(* CODESYS project sensata_common.library
   Company: Sensata Technologies
   DocFormat: reStructuredText
   Description: Library containing Sensata's high-level abstract modules that Sensata's other modules are built upon.
   Version: 1.0.0
   Placeholder: Sensata_Common
   Title: Sensata_Common

Project tree, tasks and I/O mapping:
  libraries: Tc2_Standard, 3.3.3.0 (Beckhoff Automation GmbH); Tc2_System, 3.4.25.0 (Beckhoff Automation GmbH); Tc2_Utilities, 3.3.52.0 (Beckhoff Automation GmbH); Tc3_JsonXml, * (Beckhoff Automation GmbH); Tc3_Module, 3.3.21.0 (Beckhoff Automation GmbH)
  Abstract/
    function block FB_Device [ST]: M_Abort, P_bAbortBusy, M_Connect, M_Disconnect, M_GetConnectStatus, P_bConnectBusy, P_bConnected, P_strDescription, P_strMake, P_strModel, P_strVersion, M_Disable, M_Enable, M_GetEnableStatus, P_bEnableBusy, P_bEnabled, M_GetPowerStatus, M_PowerOff, M_PowerOn, P_bPowerBusy, P_bPoweredOn, M_GetCurrentProgram, M_GetProgramState, M_LoadProgram, M_PauseProgram, M_StartProgram, M_StopProgram, P_bProgramControlBusy, P_enumProgramState, P_strCurrentProgram, M_Reset, P_bResetBusy
    function block FB_Machine [ST]: M_ResetCommands, M001_Aborting, M021_Clearing, M101_Stopping, M201_Resetting, M301_Starting, M321_Completing, M401_Holding, M421_Unholding, M501_Suspending, M521_Unsuspending, M_AbortStations, M_ClearStations, M_CompleteStations, M_HoldStations, M_ResetStations, M_StartStations, M_StopStations, M_SuspendStations, M_UnholdStations, M_UnsuspendStations, M_CheckStations, M_SetStation, P_arrStations
    function block FB_Module [ST]: M_ClearError, M_SetError, P_bError, P_strErrorMessage, P_udintErrorCode, M_Log, M_LogError, M_LogMessage, M_LogWarning, P_bLoggingEnabled, P_strUniqueId
    function block FB_StateMachine [ST]: P_bAbortable, P_bStoppable, P_enumState, M_Abort, M_Clear, M_Complete, M_Hold, M_Reset, M_Start, M_Stop, M_Suspend, M_Unhold, M_Unsuspend, A000_Aborting_Entry, A001_Aborting, A002_Aborting_Exit, M000_Aborting_Entry, M001_Aborting, M002_Aborting_Exit, A010_Aborted_Entry, A011_Aborted, A012_Aborted_Exit, M010_Aborted_Entry, M011_Aborted, M012_Aborted_Exit, A020_Clearing_Entry, A021_Clearing, A022_Clearing_Exit, M020_Clearing_Entry, M021_Clearing, M022_Clearing_Exit, A100_Stopping_Entry, A101_Stopping, A102_Stopping_Exit, M100_Stopping_Entry, M101_Stopping, M102_Stopping_Exit, A110_Stopped_Entry, A111_Stopped, A112_Stopped_Exit, M110_Stopped_Entry, M111_Stopped, M112_Stopped_Exit, A200_Resetting_Entry, A201_Resetting, A202_Resetting_Exit, M200_Resetting_Entry, M201_Resetting, M202_Resetting_Exit, A210_Idle_Entry, A211_Idle, A212_Idle_Exit, M210_Idle_Entry, M211_Idle, M212_Idle_Exit, A300_Starting_Entry, A301_Starting, A302_Starting_Exit, M300_Starting_Entry, M301_Starting, M302_Starting_Exit, A310_Execute_Entry, A311_Execute, A312_Execute_Exit, M310_Execute_Entry, M311_Execute, M312_Execute_Exit, A320_Completing_Entry, A321_Completing, A322_Completing_Exit, M320_Completing_Entry, M321_Completing, M322_Completing_Exit, A330_Complete_Entry, A331_Complete, A332_Complete_Exit, M330_Complete_Entry, M331_Complete, M332_Complete_Exit, A400_Holding_Entry, A401_Holding, A402_Holding_Exit, M400_Holding_Entry, M401_Holding, M402_Holding_Exit, A410_Held_Entry, A411_Held, A412_Held_Exit, M410_Held_Entry, M411_Held, M412_Held_Exit, A420_Unholding_Entry, A421_Unholding, A422_Unholding_Exit, M420_Unholding_Entry, M421_Unholding, M422_Unholding_Exit, A500_Suspending_Entry, A501_Suspending, A502_Suspending_Exit, M500_Suspending_Entry, M501_Suspending, M502_Suspending_Exit, A510_Suspended_Entry, A511_Suspended, A512_Suspended_Exit, M510_Suspended_Entry, M511_Suspended, M512_Suspended_Exit, A520_Unsuspending_Entry, A521_Unsuspending, A522_Unsuspending_Exit, M520_Unsuspending_Entry, M521_Unsuspending, M522_Unsuspending_Exit, A_StateMachine
    function block FB_Station [ST]: M001_Aborting, M021_Clearing, M101_Stopping, M201_Resetting, M301_Starting, M321_Completing, M401_Holding, M421_Unholding, M501_Suspending, M521_Unsuspending, M_AbortDevices, M_CheckForDeviceErrors, M_ClearDevices, M_CompleteDevices, M_HoldDevices, M_ResetDevices, M_StartDevices, M_StopDevices, M_SuspendDevices, M_UnholdDevices, M_UnsuspendDevices, M_SetDevice, P_arrDevices, M_Init, FB_exit
  Concrete/
    Obsolete/
      function block FB_DeviceTestStation_Old [ST]: M000_Aborting_Entry, M001_Aborting, M002_Aborting_Exit, M010_Aborted_Entry, M011_Aborted, M012_Aborted_Exit, M020_Clearing_Entry, M021_Clearing, M022_Clearing_Exit, M100_Stopping_Entry, M101_Stopping, M102_Stopping_Exit, M110_Stopped_Entry, M111_Stopped, M112_Stopped_Exit, M200_Resetting_Entry, M201_Resetting, M202_Resetting_Exit, M210_Idle_Entry, M211_Idle, M212_Idle_Exit, M300_Starting_Entry, M301_Starting, M302_Starting_Exit, M310_Execute_Entry, M311_Execute, M312_Execute_Exit, M320_Completing_Entry, M321_Completing, M322_Completing_Exit, M330_Complete_Entry, M331_Complete, M332_Complete_Exit, M400_Holding_Entry, M401_Holding, M402_Holding_Exit, M410_Held_Entry, M411_Held, M412_Held_Exit, M420_Unholding_Entry, M421_Unholding, M422_Unholding_Exit, M500_Suspending_Entry, M501_Suspending, M502_Suspending_Exit, M510_Suspended_Entry, M511_Suspended, M512_Suspended_Exit, M520_Unsuspending_Entry, M521_Unsuspending, M522_Unsuspending_Exit, A_DeviceTestTracking
    function block FB_DeviceController [ST]: M_Init, M00_Abort, M02_Clear, M10_Stop, M20_Reset, M30_Start, M32_Complete, M40_Hold, M42_Unhold, M50_Suspend, M52_Unsuspend
    function block FB_DeviceTestStation [ST]: A_DeviceTestTracking
    function block FB_SimpleMachine [ST]: A_Buttons, A_RunSimpleMachine, A_StopAndAbort, M011_Aborted, M111_Stopped, M211_Idle, M311_Execute, M331_Complete, M411_Held, M511_Suspended
    function block FB_SimpleStation [ST]: A_Buttons, A_RunSimpleStation, A_StopAndAbort, M011_Aborted, M111_Stopped, M211_Idle, M311_Execute, M331_Complete, M411_Held, M511_Suspended
    function block FB_StandardStation [ST]: M_AwaitCycleEnd, M_AwaitCycleStart, M_ClearUserPrompt, M_HandleException, M_ResetCycle, M_SetUserPrompt
  Enumerators/
    data type E_DeviceControllerError
    data type E_MachineError
    data type E_PackMLState
    data type E_ProgramState
    data type E_StationError
  Global Variable Lists/
    global variables GVL_Constants
  Interfaces/
    Devices/
      interface I_Abortable: M_Abort, P_bAbortBusy
      interface I_Connectable: M_Connect, M_Disconnect, M_GetConnectStatus, P_bConnectBusy, P_bConnected
      interface I_DeviceInfo: P_strDescription, P_strMake, P_strModel, P_strVersion
      interface I_Enableable: M_Disable, M_Enable, M_GetEnableStatus, P_bEnableBusy, P_bEnabled
      interface I_Powerable: M_GetPowerStatus, M_PowerOff, M_PowerOn, P_bPowerBusy, P_bPoweredOn
      interface I_Programmable: M_GetCurrentProgram, M_GetProgramState, M_LoadProgram, M_PauseProgram, M_StartProgram, M_StopProgram, P_bProgramControlBusy, P_enumProgramState, P_strCurrentProgram
      interface I_Resettable: M_Reset, P_bResetBusy
    Machines/
      interface I_MachineStationStateControl: M_AbortStations, M_ClearStations, M_CompleteStations, M_HoldStations, M_ResetStations, M_StartStations, M_StopStations, M_SuspendStations, M_UnholdStations, M_UnsuspendStations
    Modules/
      interface I_ErrorHandling: M_ClearError, M_SetError, P_bError, P_strErrorMessage, P_udintErrorCode
      interface I_Logging: M_LogError, M_LogMessage, M_LogWarning, P_bLoggingEnabled
    State Machine/
      Stateful/
        interface I_ExecuteStateOnly: M310_Execute_Entry, M312_Execute_Exit
        interface I_SimpleExecuteStateOnly: M311_Execute
        interface I_SimpleStateful
        interface I_SimpleTransitionStatesOnly: M001_Aborting, M021_Clearing, M101_Stopping, M201_Resetting, M301_Starting, M321_Completing, M401_Holding, M421_Unholding, M501_Suspending, M521_Unsuspending
        interface I_SimpleWaitingStatesOnly: M011_Aborted, M111_Stopped, M211_Idle, M331_Complete, M411_Held, M511_Suspended
        interface I_Stateful
        interface I_TransitionStatesOnly: M000_Aborting_Entry, M002_Aborting_Exit, M020_Clearing_Entry, M022_Clearing_Exit, M100_Stopping_Entry, M102_Stopping_Exit, M200_Resetting_Entry, M202_Resetting_Exit, M300_Starting_Entry, M302_Starting_Exit, M320_Completing_Entry, M322_Completing_Exit, M400_Holding_Entry, M402_Holding_Exit, M420_Unholding_Entry, M422_Unholding_Exit, M500_Suspending_Entry, M502_Suspending_Exit, M520_Unsuspending_Entry, M522_Unsuspending_Exit
        interface I_WaitingStatesOnly: M010_Aborted_Entry, M012_Aborted_Exit, M110_Stopped_Entry, M112_Stopped_Exit, M210_Idle_Entry, M212_Idle_Exit, M310_Execute_Entry, M312_Execute_Exit, M330_Complete_Entry, M332_Complete_Exit, M410_Held_Entry, M412_Held_Exit, M510_Suspended_Entry, M512_Suspended_Exit
      interface I_StateControl: M_Abort, M_Clear, M_Complete, M_Hold, M_Reset, M_Start, M_Stop, M_Suspend, M_Unhold, M_Unsuspend
    Stations/
      interface I_StationDeviceControl: M_AbortDevices, M_ClearDevices, M_CompleteDevices, M_HoldDevices, M_ResetDevices, M_StartDevices, M_StopDevices, M_SuspendDevices, M_UnholdDevices, M_UnsuspendDevices
  Project Information/
    function F_GetCompany [ST]
    function F_GetTitle [ST]
    function F_GetVersion [ST]
  Structs/
    data type ST_Prompt
  Types/
    data type T_MachineStationArray
    data type T_StationDeviceArray
  Version/
    global variables Global_Version
*)

// Enumerators/E_DeviceControllerError
{attribute 'qualified_only'}
{attribute 'strict'}
{attribute 'qualified_only'}
TYPE E_DeviceControllerError :
(
	None := 0,
	ClearError := 0200,
	StopError := 1000,
	ResetError := 2000,
	StartError := 3000,
	CompleteError := 3200,
	HoldError := 4000,
	UnholdError := 4200,
	SuspendError := 5000,
	UnsuspendError := 5200
) UDINT;
END_TYPE

// Enumerators/E_MachineError
{attribute 'qualified_only'}
{attribute 'strict'}
TYPE E_MachineError :
(
	None := 0,
	
	StationError := 100
) UDINT;
END_TYPE

// Enumerators/E_PackMLState
(* Represents all possible PackML states. *)
{attribute 'qualified_only'}
{attribute 'strict'}
{attribute 'to_string'}
TYPE E_PackMLState :
(
	None := -1,
	Aborting := 00, 
	Aborted := 01,
	Clearing := 02,
	Stopping := 10,
	Stopped := 11,
	Resetting := 20,
	Idle := 21, 
	Starting := 30,
	Execute := 31,
	Completing := 32,
	Complete := 33,
	Holding := 40,
	Held := 41,
	Unholding := 42,
	Suspending := 50,
	Suspended := 51,
	Unsuspending := 52
) := None;
END_TYPE

// Enumerators/E_ProgramState
(*
The possible states for a program loaded on a device.
*)
{attribute 'qualified_only'}
{attribute 'strict'}
{attribute 'to_string'}
TYPE E_ProgramState :
(
	(* The unknown state means that the current program state is not known.
		This is the default enumerator state. *)
	Unknown := 0,
	
	(* A program that is stopped means that, when started, the program would begin
		from the start. Going from the Running state to the Stopped state or from
		the Paused state to the Stopped state will reset the program execution
		back to the beginning. *)
	Stopped,
	
	(* A program in the running state is actively executing. Going from the
		Stopped state to the Running state will begin execution from the
		beginning of the program, and going from the Paused state to the
		Running state will continue execution from whichever point it was
		at when the transition from Running to Paused occurred.*)
	Running,
	
	(* A program that is paused is not executing, but is also not reset to the
		start. When going from the Running state to the Paused state, the
		program execution is held in the state it was in when the transition
		occurred. *)
	Paused
);
END_TYPE

// Enumerators/E_StationError
{attribute 'qualified_only'}
{attribute 'strict'}
(*
Errors for use in FB_Station
*)
TYPE E_StationError :
(
	None			:= 000000000,
	
	DeviceError		:= 301000000
) UDINT;
END_TYPE

// Structs/ST_Prompt
TYPE ST_Prompt :
STRUCT
	(* Code for this prompt message. *)
	udintCode: UDINT;
	(* Default message text (for debug and if localization not used) *)
	strMessage: T_MaxString;
END_STRUCT
END_TYPE

// Types/T_MachineStationArray
(* Alias for an array of pointers to stations. *)
TYPE T_MachineStationArray : 
	ARRAY[1..GVL_Constants.uintMAX_MACHINE_STATION_COUNT] 
		OF POINTER TO FB_Station;
END_TYPE

// Types/T_StationDeviceArray
(* Alias for an array of pointers to devices. *)
TYPE T_StationDeviceArray :
	ARRAY[1..GVL_Constants.uintMAX_STATION_DEVICE_COUNT]
		OF POINTER TO FB_DeviceController;
END_TYPE

// Global Variable Lists/GVL_Constants
{attribute 'qualified_only'}
VAR_GLOBAL CONSTANT
	uintMAX_STATION_DEVICE_COUNT : UINT := 32;
	uintMAX_MACHINE_STATION_COUNT : UINT := 32;
END_VAR

// Version/Global_Version
{attribute 'TcGenerated'}
{attribute 'no-analysis'}
{attribute 'linkalways'}
// This function has been automatically generated from the project information.
VAR_GLOBAL CONSTANT
	{attribute 'const_non_replaced'}
	stLibVersion_Sensata_Common : ST_LibVersion := (iMajor := 1, iMinor := 0, iBuild := 0, iRevision := 0, nFlags := 0, sVersion := '1.0.0');
END_VAR

// Abstract/FB_Device
(*
===============================================================================
Device
===============================================================================
:Contact: Kevin Sanita <ksanita@sensata.com>
:Last Edited: December 2021

:Description: Parent class for all devices in the Sensata libraries.

:Notes:
* Devices are defined as physical objects that the PAC must control or communicate with.
* All children of this Device class should implement ``I_DeviceInfo`` to easily import the required properties.
* Ensure the device properties are properly implemented and kept up to date if a device is updated.

:Change Log:
- **December 2021** Initial version
*)
{attribute 'hide_all_locals'}
FUNCTION_BLOCK ABSTRACT FB_Device EXTENDS FB_Module 
	IMPLEMENTS 
		I_DeviceInfo, // Device information
		I_Abortable, // Some devices may need to perform specific tasks when aborted
		I_Connectable, // Connecting and disconnecting is a common functionality of devices
		I_Enableable, // Many devices can be enabled/disabled without necessarily changing state
		I_Powerable, // Many devices need a specific command in order to energize
		I_Programmable, // Managing programs is a common functionality of devices with internal logic
		I_Resettable // Devices often need a reset command to clear any errors
VAR_INPUT		
END_VAR
VAR_OUTPUT
END_VAR
VAR
	dev_bConnected: BOOL; // TRUE if the device is connected
	dev_bEnabled: BOOL; // TRUE if the device is enabled
	dev_enumProgramState: E_ProgramState; // Current control state
	dev_bPoweredOn: BOOL; // TRUE if the device is powered on
	dev_strCurrentProgram: STRING(255); // Current program
END_VAR

(* Performs tasks that should be performed when the device is aborted. *)
METHOD M_Abort : BOOL
M_Abort := TRUE;
THIS^.M_LogWarning('M_Abort not implemented!');

IF NOT THIS^.P_bError THEN
	THIS^.M_SetError(16#FFFF, 'Aborted!');
END_IF
END_METHOD

(* True while aborting, false otherwise. *)
PROPERTY P_bAbortBusy : BOOL
GET
P_bAbortBusy := FALSE;
END_GET
END_PROPERTY

(* Connect to the device. *)
METHOD M_Connect : BOOL
dev_bConnected := TRUE;
M_Connect := TRUE;
THIS^.M_LogWarning('M_Connect not implemented!');
END_METHOD

(* Disconnect from the camera. *)
METHOD M_Disconnect : BOOL
dev_bConnected := FALSE;
M_Disconnect := TRUE;
THIS^.M_LogWarning('M_Disconnect not implemented!');
END_METHOD

(* Get the device connection status. *)
METHOD M_GetConnectStatus : BOOL
VAR_OUTPUT
	(* TRUE if the device is connected, FALSE otherwise. *)
	bConnected	: BOOL;
END_VAR
bConnected := THIS^.dev_bConnected;
M_GetConnectStatus := TRUE;
END_METHOD

(* TRUE while the device is connecting or disconnecting. *)
PROPERTY P_bConnectBusy : BOOL
GET
P_bConnectBusy := FALSE;
END_GET
END_PROPERTY

(* TRUE if the camera is connected. *)
PROPERTY P_bConnected : BOOL
GET
P_bConnected := dev_bConnected;
END_GET
END_PROPERTY

(*
A brief description of the device.
*)
PROPERTY P_strDescription : T_MaxString
GET
END_GET
END_PROPERTY

(*
The manufacturer of the device.
*)
PROPERTY P_strMake : T_MaxString
GET
END_GET
END_PROPERTY

(*
The model name or ID of the device.
*)
PROPERTY P_strModel : T_MaxString
GET
END_GET
END_PROPERTY

(*
The version(s) of the device that the function block supports.
*)
PROPERTY P_strVersion : T_MaxString
GET
END_GET
END_PROPERTY

(* Disable the device. *)
METHOD M_Disable : BOOL
dev_bEnabled := FALSE;
M_Disable := TRUE;
THIS^.M_LogWarning('M_Disable is not implemented!');
END_METHOD

(* Enable the device *)
METHOD M_Enable : BOOL
dev_bEnabled := TRUE;
M_Enable := TRUE;
THIS^.M_LogWarning('M_Enable is not implemented!');
END_METHOD

(* Get the current enable status of the device. *)
METHOD M_GetEnableStatus : BOOL
VAR_OUTPUT
	bEnabled	: BOOL;
END_VAR
bEnabled := THIS^.dev_bEnabled;
M_GetEnableStatus := TRUE;
END_METHOD

(* TRUE while the device is busy enabling or disabling. *)
PROPERTY P_bEnableBusy : BOOL
GET
END_GET
END_PROPERTY

(* TRUE if the device is enabled. *)
PROPERTY P_bEnabled : BOOL
GET
P_bEnabled := dev_bEnabled;
END_GET
END_PROPERTY

(* Gets the current power status of the device. *)
METHOD M_GetPowerStatus : BOOL
VAR_OUTPUT
	bPoweredOn	: BOOL;
END_VAR
bPoweredOn := THIS^.dev_bPoweredOn;
M_GetPowerStatus := TRUE;
END_METHOD

(*
Power off the device or module
*)
METHOD M_PowerOff : BOOL
dev_bPoweredOn := FALSE;
M_PowerOff := TRUE;
THIS^.M_LogWarning('M_PowerOff is not implemented!');
END_METHOD

(*
Power on the device or module.
*)
METHOD M_PowerOn : BOOL
dev_bPoweredOn := TRUE;
M_PowerOn := TRUE;
THIS^.M_LogWarning('M_PowerOn is not implemented!');
END_METHOD

(* TRUE while the device is powering on or off. *)
PROPERTY P_bPowerBusy : BOOL
GET
P_bPowerBusy := FALSE;
END_GET
END_PROPERTY

(*
TRUE if the module or device is powered on.
*)
PROPERTY P_bPoweredOn : BOOL
GET
P_bPoweredOn := dev_bPoweredOn;
END_GET
END_PROPERTY

(* Gets the program currently loaded on the device. *)
METHOD M_GetCurrentProgram : BOOL
VAR_OUTPUT
	strCurrentProgram	: Tc2_System.T_MaxString;
END_VAR
strCurrentProgram := THIS^.dev_strCurrentProgram;
M_GetCurrentProgram := TRUE;
END_METHOD

(* Gets the current control state. *)
METHOD M_GetProgramState : BOOL
VAR_OUTPUT
	enumProgramState	: E_ProgramState;
END_VAR
enumProgramState := THIS^.dev_enumProgramState;
M_GetProgramState := TRUE;
END_METHOD

(* Load a new program. *)
METHOD M_LoadProgram : BOOL
VAR_INPUT
END_VAR
dev_strCurrentProgram := '';
M_LoadProgram := TRUE;
THIS^.M_LogWarning('M_LoadProgram not implemented!');
END_METHOD

(* Pauses the camera program. *)
METHOD M_PauseProgram : BOOL
dev_enumProgramState := E_ProgramState.Paused;
M_PauseProgram := TRUE;
THIS^.M_LogWarning('M_PauseProgram not implemented!');
END_METHOD

(* Starts the camera program. *)
METHOD M_StartProgram : BOOL
dev_enumProgramState := E_ProgramState.Running;
M_StartProgram := TRUE;
THIS^.M_LogWarning('M_StartProgram not implemented!');
END_METHOD

(* Stops the camera program. *)
METHOD M_StopProgram : BOOL
dev_enumProgramState := E_ProgramState.Stopped;
M_StopProgram := TRUE;
THIS^.M_LogWarning('M_StopProgram not implemented!');
END_METHOD

(*
TRUE while a program is being loaded
*)
PROPERTY P_bProgramControlBusy : BOOL
GET
P_bProgramControlBusy := FALSE;
END_GET
END_PROPERTY

(* Current device program state. *)
PROPERTY P_enumProgramState : E_ProgramState
GET
P_enumProgramState := dev_enumProgramState;
END_GET
END_PROPERTY

(* Current program. *)
PROPERTY P_strCurrentProgram : Tc2_System.T_MaxString
GET
P_strCurrentProgram := dev_strCurrentProgram;
END_GET
END_PROPERTY

(* Resets the device and clears any external errors. *)
METHOD M_Reset : BOOL
M_Reset := TRUE;
THIS^.M_ClearError();
THIS^.M_LogWarning('M_Reset not implemented!');
END_METHOD

(* Stays high while module is resetting. *)
PROPERTY P_bResetBusy : BOOL
GET
P_bResetBusy := FALSE;
END_GET
END_PROPERTY

END_FUNCTION_BLOCK

// Interfaces/Devices/I_DeviceInfo
(*
===============================================================================
Device Information
===============================================================================

:Description: Contains the standard properties of the Device function block for easier implementation.

*)
INTERFACE I_DeviceInfo

PROPERTY P_strDescription : T_MaxString
GET
END_GET
END_PROPERTY

PROPERTY P_strMake : T_MaxString
GET
END_GET
END_PROPERTY

PROPERTY P_strModel : T_MaxString
GET
END_GET
END_PROPERTY

PROPERTY P_strVersion : T_MaxString
GET
END_GET
END_PROPERTY

END_INTERFACE

// Abstract/FB_Module
(*
===============================================================================
Module
===============================================================================
:Contact: Kevin Sanita <ksanita@sensata.com>
:Last Edited: December 2021

:Description: All function blocks in Sensata libraries must derive from this. Handles basic functions like errors and logging. 

:Notes:
* You can use ``M_LogError``, ``M_LogWarning``, and ``M_LogMessage`` to output string messages to the "Error list" in Visual Studio
* ``M_SetError`` and ``M_ClearError`` can be used to set an error with a specified error code and message and then clear said error.
* You can use ``P_bError``, ``P_strErrorMessage`` and ``P_udintErrorCode`` to access error information.

:Change Log:
- **December 2021** Initial version

*)
FUNCTION_BLOCK ABSTRACT FB_Module
	IMPLEMENTS
		I_ErrorHandling, // All modules have error handling
		I_Logging // All modules have logging
VAR_INPUT CONSTANT
	in_strUniqueId : T_MaxString; (* A unique name for this function block to be used in logging. *)
	in_bDisableLogging: BOOL; (* Set TRUE to disable all logging. *)
END_VAR
VAR_OUTPUT
END_VAR
VAR
	mod_bError : BOOL; (* TRUE if there is an error. *)
	mod_udintErrorCode : UDINT; (* 0 if no error, error code otherwise. Refer to module-specific documentation for code meaning. *)
	mod_strErrorMessage : T_MaxString; (* Blank if no error, error message otherwise. *)
	mod_bLoggingEnabled: BOOL := TRUE; (* Enables and disabled logging. *)
END_VAR

(*
Clears the current error. Sets P_bError to false, P_strErrorMessage to blank, and P_udintErrorCode to zero.
*)
METHOD M_ClearError : BOOL
IF THIS^.mod_bError THEN
	THIS^.M_LogMessage('Error cleared.');
END_IF

THIS^.mod_bError := FALSE;
THIS^.mod_udintErrorCode := 0;
THIS^.mod_strErrorMessage := '';

M_ClearError := TRUE;
END_METHOD

(*
Sets an error with the given code and message.
*)
METHOD M_SetError : BOOL
VAR_INPUT
	udintErrorCode : UDINT; (* Error codes are specific to the concrete modules. Check documentation of the module for error code meaning. *)
	strErrorMessage : T_MaxString; (* Error messages should be short, but descriptive enough to still be useful. *)
END_VAR
// If there is not already an error set or error code or message is different,
// update the values and print to log
IF (NOT mod_bError) 
		OR (mod_udintErrorCode <> udintErrorCode)
		OR (mod_strErrorMessage <> strErrorMessage) THEN
	THIS^.mod_bError := TRUE;
	THIS^.mod_udintErrorCode := udintErrorCode;
	THIS^.mod_strErrorMessage := strErrorMessage;
	THIS^.M_LogError(strErrorMessage);
END_IF
END_METHOD

(*
TRUE if there is an error, FALSE otherwise.
*)
PROPERTY P_bError : BOOL
GET
P_bError := mod_bError;
END_GET
END_PROPERTY

(*
A description of the current error. Will be blank if no error.
*)
PROPERTY P_strErrorMessage : Tc2_System.T_MaxString
GET
P_strErrorMessage := mod_strErrorMessage;
END_GET
END_PROPERTY

(*
The ID of the current error. Review module-specific documentation for meaning of error codes. Will be 0 if no error.
*)
PROPERTY P_udintErrorCode : UDINT
GET
P_udintErrorCode := mod_udintErrorCode;
END_GET
END_PROPERTY

METHOD PRIVATE M_Log : BOOL
VAR_INPUT
	strMessage : T_MaxString;
	dwordMsgCtrlMask : DWORD;
END_VAR
VAR
	fbFormat: FB_FormatString;
END_VAR
// If logging is enabled, print to ADS log
IF NOT in_bDisableLogging THEN
	// Format the message with the unique ID
	fbFormat(
		sFormat:= '%s --- %s', 
		arg1:= F_STRING(in_strUniqueId), 
		arg2:= F_STRING(strMessage));
	
	// Return false if there was a format error
	IF fbFormat.bError THEN
		M_Log := FALSE;
	ELSE
		// Log the message to ADS
		ADSLOGSTR(
			msgCtrlMask:= dwordMsgCtrlMask,
			msgFmtStr:= '%s',
			strArg:= fbFormat.sOut);
		M_Log := TRUE;
	END_IF
// If logging is not enabled, don't do anything
ELSE
	M_Log := TRUE;
END_IF
END_METHOD

(*
Prints an error message to the Error List in Visual Studio.
*)
METHOD M_LogError : BOOL
VAR_INPUT
	strMessage : T_MaxString;
END_VAR
M_LogError := M_Log(strMessage, ADSLOG_MSGTYPE_ERROR OR ADSLOG_MSGTYPE_LOG);
END_METHOD

(*
Outputs a message to the Error List in Visual Studio
*)
METHOD M_LogMessage : BOOL
VAR_INPUT
	strMessage : T_MaxString;
END_VAR
M_LogMessage := M_Log(strMessage, ADSLOG_MSGTYPE_HINT OR ADSLOG_MSGTYPE_LOG);
END_METHOD

(*
Outputs a warning message to the Error List in Visual Studio
*)
METHOD M_LogWarning : BOOL
VAR_INPUT
	strMessage : T_MaxString;
END_VAR
M_LogWarning := M_Log(strMessage, ADSLOG_MSGTYPE_WARN OR ADSLOG_MSGTYPE_LOG);
END_METHOD

(* TRUE when ADS logging is enabled, false otherwise. *)
PROPERTY P_bLoggingEnabled : BOOL
GET
P_bLoggingEnabled := NOT in_bDisableLogging;
END_GET
END_PROPERTY

PROPERTY P_strUniqueId : T_MaxString
GET
P_strUniqueId := in_strUniqueId;
END_GET
END_PROPERTY

END_FUNCTION_BLOCK

// Interfaces/Modules/I_ErrorHandling
INTERFACE I_ErrorHandling

(*
Clears the current error. Sets P_bError to false, P_strErrorMessage to blank, and P_udintErrorCode to zero.
*)
METHOD M_ClearError : BOOL
END_METHOD

(*
Sets an error with the given code and message.
*)
METHOD M_SetError : BOOL
VAR_INPUT
	udintErrorCode : UDINT; (* Error codes are specific to the concrete modules. Check documentation of the module for error code meaning. *)
	strErrorMessage : T_MaxString; (* Error messages should be short, but descriptive enough to still be useful. *)
END_VAR
END_METHOD

(*
TRUE if there is an error, FALSE otherwise.
*)
PROPERTY P_bError : BOOL
GET
END_GET
END_PROPERTY

(*
A description of the current error. Will be blank if no error.
*)
PROPERTY P_strErrorMessage : Tc2_System.T_MaxString
GET
END_GET
END_PROPERTY

(*
The ID of the current error. Review module-specific documentation for meaning of error codes. Will be 0 if no error.
*)
PROPERTY P_udintErrorCode : UDINT
GET
END_GET
END_PROPERTY

END_INTERFACE

// Interfaces/Modules/I_Logging
INTERFACE I_Logging

(*
Prints an error message to the Error List in Visual Studio.
*)
METHOD M_LogError : BOOL
VAR_INPUT
	strMessage : T_MaxString;
END_VAR
END_METHOD

(*
Outputs a message to the Error List in Visual Studio
*)
METHOD M_LogMessage : BOOL
VAR_INPUT
	strMessage : T_MaxString;
END_VAR
END_METHOD

(*
Outputs a warning message to the Error List in Visual Studio
*)
METHOD M_LogWarning : BOOL
VAR_INPUT
	strMessage : T_MaxString;
END_VAR
END_METHOD

(* TRUE when ADS logging is enabled, false otherwise. *)
PROPERTY P_bLoggingEnabled : BOOL
GET
END_GET
END_PROPERTY

END_INTERFACE

// Interfaces/Devices/I_Abortable
(*
===============================================================================
Abortable
===============================================================================

:Description: Implements the ability to quickly and safely abort the device.
*)
INTERFACE I_Abortable

(* This method should rapidly but safely abort the device and set an error
	indicating that the device has been aborted. Method should return TRUE
	once successfully aborted and false otherwise. *)
METHOD M_Abort : BOOL
VAR_INPUT
END_VAR
END_METHOD

(* This property should be TRUE while any method in this interface is actively
	executing, or FALSE otherwise. *)
PROPERTY P_bAbortBusy : BOOL
GET
END_GET
END_PROPERTY

END_INTERFACE

// Interfaces/Devices/I_Connectable
(*
===============================================================================
Connectable
===============================================================================

:Description: Implements the ability to send explicit connect and disconnect
	commands to the device.
*)
INTERFACE I_Connectable

(* This method should establish any external connections required to use the
	functions of the device, and return TRUE and set P_bConnected to TRUE once
	connected. *)
METHOD M_Connect : BOOL
VAR_INPUT
END_VAR
END_METHOD

(* This method should break any connections established by M_Connect. It should
	immediately set P_bConnected to false unless all connections are known to
	be still active, and return TRUE once those connections are all fully
	disconnected. *)
METHOD M_Disconnect : BOOL
VAR_INPUT
END_VAR
END_METHOD

(* This method should explicitly check the connection status of the device.
	Once the connection status is known, this method should return TRUE.
	If this method fails, P_bConnected should be set to FALSE since the device
	is not absolutely known to still be connected. *)
METHOD M_GetConnectStatus : BOOL
VAR_INPUT
END_VAR
VAR_OUTPUT
	(* This should return TRUE if all connections required to make the device
		function properly are known to be connected, and FALSE otherwise. *)
	bConnected : BOOL;
END_VAR
END_METHOD

(* This property should be TRUE while any method in this interface is actively
	executing, or FALSE otherwise. *)
PROPERTY P_bConnectBusy : BOOL
GET
END_GET
END_PROPERTY

(* This should be set to TRUE if M_Connect is successful or M_GetConnectStatus
	determines the device to be connected, and set to FALSE if M_Disconnect is
	called at all, M_GetConnectStatus fails, or M_GetConnectStatus determines
	the device to be not connected. *)
PROPERTY P_bConnected : BOOL
GET
END_GET
END_PROPERTY

END_INTERFACE

// Interfaces/Devices/I_Enableable
(*
===============================================================================
Enableable
===============================================================================

:Description: Interface that implements the ability for the device to enable to
	(and disable from) a ready-to-start state from an energized state.

*)
INTERFACE I_Enableable

(* This method should return to the device to the state it was prior to being
	enabled. P_bEnabled should be immediately set to false unless the status of
	the device is explicitly known to still be enabled. After being disabled,
	the device should typically be unable to perform process steps. Once
	successfully disabled, this method should return TRUE. *)
METHOD M_Disable : BOOL
VAR_INPUT
END_VAR
END_METHOD

(* This method should perform any tasks that must be performed after a device
	is energized, but prior to the device being used in a process, and then
	return TRUE and set P_bEnabled to TRUE once those tasks are completed. *)
METHOD M_Enable : BOOL
VAR_INPUT
END_VAR
END_METHOD

(* This method should explicitly check the enable status of the device.
	Once the enable status is known, this method should return TRUE.
	If this method fails, P_bEnabled should be set to FALSE since the device
	is not absolutely known to still be enabled. *)
METHOD M_GetEnableStatus : BOOL
VAR_INPUT
END_VAR
VAR_OUTPUT
	(* This should return TRUE if the device is explicitly known to be
		enabled, or FALSE otherwise. *)
	bEnabled : BOOL;
END_VAR
END_METHOD

(* This property should be TRUE while any method in this interface is actively
	executing, or FALSE otherwise. *)
PROPERTY P_bEnableBusy : BOOL
GET
END_GET
END_PROPERTY

(* This should be set to TRUE if M_Enable is successful or M_GetEnableStatus
	determines the device to be enabled, and set to FALSE if M_Disable is
	called at all, M_GetEnableStatus fails, or M_GetEnableStatus determines
	the device to be not enabled. *)
PROPERTY P_bEnabled : BOOL
GET
END_GET
END_PROPERTY

END_INTERFACE

// Interfaces/Devices/I_Powerable
(*
===============================================================================
Powerable
===============================================================================

:Description: Interface that implements the ability to energize and de-energize
	a device. 

*)
INTERFACE I_Powerable

(* This method should explicitly check the power status of the device.
	Once the power status is known, this method should return TRUE.
	If this method fails, P_bPoweredOn should be set to FALSE since the device
	is not absolutely known to still be powered on. *)
METHOD M_GetPowerStatus : BOOL
VAR_INPUT
END_VAR
VAR_OUTPUT
	(* This should return TRUE if the device is explicitly known to be
		powered on, or FALSE otherwise. *)
	bPoweredOn : BOOL;
END_VAR
END_METHOD

(* This method should de-energize the device and then return TRUE once
	successful. P_bPoweredOn should be set to FALSE immediately when this is
	called unless the device is explicitly known to still be powered on. *)
METHOD M_PowerOff : BOOL
VAR_INPUT
END_VAR
END_METHOD

(* This method should energize the device and then return TRUE and set
	P_bPoweredOn to TRUE once successful. *)
METHOD M_PowerOn : BOOL
VAR_INPUT
END_VAR
END_METHOD

(* This property should be TRUE while any method in this interface is actively
	executing, or FALSE otherwise. *)
PROPERTY P_bPowerBusy : BOOL
GET
END_GET
END_PROPERTY

(* This should be set to TRUE if M_PowerOn is successful or if M_GetPowerStatus
	determines that the device is powered on. Otherwise, this should be FALSE. *)
PROPERTY P_bPoweredOn : BOOL
GET
END_GET
END_PROPERTY

END_INTERFACE

// Interfaces/Devices/I_Programmable
(*
===============================================================================
Programmable
===============================================================================

:Description: Interface that implements the ability to manage devices that have
	internally-defined execution programs that can be loaded and/or controlled
	by an external source.

:Change Log:
* June 2022 - Change P_bProgramLoading to P_bProgramBusy
*)
INTERFACE I_Programmable

(* This method should explicitly get the current program loaded on the device.
	If the current program is successfully gotten, this method should return
	TRUE and set P_strCurrentProgram and strCurrentProgram to the gotten
	program name. If this method fails, both should be set to empty strings. *)
METHOD M_GetCurrentProgram : BOOL
VAR_INPUT
END_VAR
VAR_OUTPUT
	(* This should be set to the name of the currently loaded program if
		the method was successful, or a blank string otherwise. *)
	strCurrentProgram : T_MaxString;
END_VAR
END_METHOD

(* This method should explicitly check the program state of the device.
	Once the program state is known, this method should return TRUE and set
	P_enumProgramState and enumProgramState to the relevant E_ProgramState
	value, else it should set both to E_ProgramState.Unknown. *)
METHOD M_GetProgramState : BOOL
VAR_INPUT
END_VAR
VAR_OUTPUT
	(* If the program state is successfully gotten, this should be set to
		the relevant E_ProgramState value. If this method fails, this should
		be set to E_ProgramState.Unknown. *)
	enumProgramState : E_ProgramState;
END_VAR
END_METHOD

(* This method should load a new program onto the device, and then return TRUE
	once program loading is completed. Once this method begins the program loading
	process, P_strCurrentProgram should be cleared unless it is still explicitly
	known to be loaded. *)
METHOD M_LoadProgram : BOOL
VAR_INPUT
END_VAR
END_METHOD

(* This program should move to the program state from whatever state it was in
	to the Paused state, and then return TRUE once successful. If the program
	state is Stopped, this method should return TRUE but keep the current state
	as Stopped, since Paused at the beginning at the program is equivalent to
	being Stopped. *)
METHOD M_PauseProgram : BOOL
VAR_INPUT
END_VAR
END_METHOD

(* This should move the program state from whatever state it is in to the
	Running state, and then return TRUE once successful. Starting from the
	Paused state should always continue execution from whatever point the
	program was at when the program was initially paused. *)
METHOD M_StartProgram : BOOL
VAR_INPUT
END_VAR
END_METHOD

(* This should change the program state from whatever state it was in to the
	Stopped state and then return TRUE. Moving to the Stopped state should
	always reset the program execution back to the beginning. *)
METHOD M_StopProgram : BOOL
VAR_INPUT
END_VAR
END_METHOD

(* This property should be TRUE while any method in this interface is actively
	executing, or FALSE otherwise. *)
PROPERTY P_bProgramControlBusy : BOOL
GET
END_GET
END_PROPERTY

(* The current E_ProgramState value of the device. This should be reset to
	E_ProgramState.Unknown if any methods in this interface interact with the
	device but fail. *)
PROPERTY P_enumProgramState : E_ProgramState
GET
END_GET
END_PROPERTY

(* The value of the currently loaded program. This should only be set by
	M_LoadProgram or M_GetCurrentProgram, and set to a blank string if either
	fail. *)
PROPERTY P_strCurrentProgram : T_MaxString
GET
END_GET
END_PROPERTY

END_INTERFACE

// Interfaces/Devices/I_Resettable
(*
===============================================================================
Resettable
===============================================================================

:Description: Interface that implements the ability to reset the device from a
	faulted state back to a ready-to-energize state.


*)
INTERFACE I_Resettable

(* This should clear any errors on the device and bring it to a state where
	it is ready to be energized or otherwise activated. *)
METHOD M_Reset : BOOL
VAR_INPUT
END_VAR
END_METHOD

(* This property should be TRUE while any method in this interface is actively
	executing, or FALSE otherwise. *)
PROPERTY P_bResetBusy : BOOL
GET
END_GET
END_PROPERTY

END_INTERFACE

// Abstract/FB_Machine
(*
===============================================================================
Machine
===============================================================================
:Contact: Kevin Sanita <ksanita@sensata.com>
:Last Edited: March 2022

:Description: Represents a machine, which is a collection of stations that must be synchronized

:Notes:
* Stations are able to implement state machines. To implement a state machine, implement I_Stateful
* In order for a state machine to run, THIS^.A_StateMachine must be called in the function block body.

:Change Log:
- **March 2022** Initial version
- **July 2022** Updating station state controls
*)
FUNCTION_BLOCK FB_Machine EXTENDS FB_StateMachine 
	IMPLEMENTS
		I_MachineStationStateControl, // Controls stations
		I_SimpleTransitionStatesOnly // Has some basic default implementations
VAR_INPUT
END_VAR
VAR_OUTPUT
END_VAR
VAR
	mac_arrStations : T_MachineStationArray;
	mac_intAbortStationsStep: INT;
	mac_intClearStationsStep: INT;
	mac_intCompleteStationsStep: INT;
	mac_intHoldStationsStep: INT;
	mac_intResetStationsStep: INT;
	mac_intStartStationsStep: INT;
	mac_intStopStationsStep: INT;
	mac_intSuspendStationsStep: INT;
	mac_intUnholdStationsStep: INT;
	mac_intUnsuspendStationsStep: INT;
END_VAR

(* Resets all state step numbers. *)
METHOD PRIVATE M_ResetCommands : BOOL
VAR_INPUT
END_VAR
mac_intAbortStationsStep :=0;
mac_intClearStationsStep :=0;
mac_intCompleteStationsStep :=0;
mac_intHoldStationsStep :=0;
mac_intResetStationsStep :=0;
mac_intStartStationsStep :=0;
mac_intStopStationsStep :=0;
mac_intSuspendStationsStep :=0;
mac_intUnholdStationsStep :=0;
mac_intUnsuspendStationsStep :=0;

M_ResetCommands := TRUE;
END_METHOD

(* The 'Aborting' state can be entered at any time while within the 'abortable'
section of the state machine. It is typically entered in response to an 'Abort'
command or a critical fault. The logic should safely but rapidly bring the
components of the module to a stop while maintaining as much information about
the pre-abort scenario as possible. *)
METHOD M001_Aborting : BOOL
VAR_OUTPUT
	(* This should be set to true once all components of the module have safely
	come to a stop. Once set to true, the state machine will move to the
	'Aborted' state. *)
	bAborted	: BOOL;
END_VAR
bAborted := THIS^.M_AbortStations();
END_METHOD

(* This state should clear any faults and reset any safety features related
to the module, as well as perform actions similar to the 'Stopping' state
if they were not already performed while aborting. *)
METHOD M021_Clearing : BOOL
VAR_OUTPUT
	(* This should be set to true once the safety state of all module
	components are reset and all errors are cleared. *)
	bCleared	: BOOL;
	(* This should be set to true if a potentially hazardous error or a safety
	fault has occurred in any tasks. Once set to true, the state machine will
	move to the 'Aborting' state. *)
	bAbort	: BOOL;
END_VAR
VAR_INST
	bErrorCleared: BOOL;
END_VAR
IF NOT bErrorCleared THEN
	bErrorCleared := TRUE;
	THIS^.M_ClearError();
END_IF
bCleared := THIS^.M_ClearStations();
IF THIS^.P_bError THEN
	bAbort := TRUE;
	bErrorCleared := FALSE;
ELSIF bCleared THEN
	bErrorCleared := FALSE;
END_IF
END_METHOD

(* This state can be entered from anywhere within the 'stoppable' group of
states. This state should safely bring the components of the module to a
controlled stop and then move to the 'Stopped' state once completed. *)
METHOD M101_Stopping : BOOL
VAR_OUTPUT
	(* This should be set to true once all relevant components have come to a
	controlled stop. Once set to true, the state machine will move to the
	'Stopped' state. *)
	bStopped	: BOOL;
	(* This should be set to true if a potentially hazardous error or a safety
	fault has occurred in any tasks. Once set to true, the state machine will
	move to the 'Aborting' state. *)
	bAbort	: BOOL;
END_VAR
IF THIS^.P_bError THEN
	bAbort := TRUE;
ELSE
	bStopped := THIS^.M_StopStations();
END_IF
END_METHOD

(* This state should place the module and all of its components into a safe
energized idle state where it will wait for a start command. Once all tasks are
complete, it will move to the 'Idle' state. No external movement should occur
as a result of this state. *)
METHOD M201_Resetting : BOOL
VAR_OUTPUT
	(* Set this to true once the module is energized and ready to start.
	Once set to true, the state machine will move to the 'Idle' state. *)
	bIdle	: BOOL;
	(* This should be set to true if an external source requests that the module
	exit its current state and come to a controlled stop. Once set to true, the
	state machine will move to the 'Stopping' state. *)
	bStop	: BOOL;
	(* This should be set to true if a potentially hazardous error or a safety
	fault has occurred in any tasks. Once set to true, the state machine will
	move to the 'Aborting' state. *)
	bAbort	: BOOL;
END_VAR
IF THIS^.P_bError THEN
	bAbort := TRUE;
ELSE
	bIdle := THIS^.M_ResetStations();
END_IF
END_METHOD

(* This state should make any final preparations needed for the 'Execute' state
prior to entering the 'Execute' state. *)
METHOD M301_Starting : BOOL
VAR_OUTPUT
	(* This should be set to true once the module and its components are fully
	prepared for process execution. Once set to true, the state machine will
	move to the 'Execute' state. *)
	bStarted	: BOOL;
	(* This should be set to true if an external source requests that the module
	exit its current state and come to a controlled stop. Once set to true, the
	state machine will move to the 'Stopping' state. *)
	bStop	: BOOL;
	(* This should be set to true if a potentially hazardous error or a safety
	fault has occurred in any tasks. Once set to true, the state machine will
	move to the 'Aborting' state. *)
	bAbort	: BOOL;
END_VAR
IF THIS^.P_bError THEN
	bAbort := TRUE;
ELSE
	bStarted := THIS^.M_StartStations();
END_IF
END_METHOD

(* This state will perform any post-execution tasks prior to moving to the
'Completed' state. *)
METHOD M321_Completing : BOOL
VAR_OUTPUT
	(* Move to the Complete state*)
	bCompleted	: BOOL;
	(* This should be set to true if an external source requests that the module
	exit its current state and come to a controlled stop. Once set to true, the
	state machine will move to the 'Stopping' state. *)
	bStop	: BOOL;
	(* This should be set to true if a potentially hazardous error or a safety
	fault has occurred in any tasks. Once set to true, the state machine will
	move to the 'Aborting' state. *)
	bAbort	: BOOL;
END_VAR
IF THIS^.P_bError THEN
	bAbort := TRUE;
ELSE
	bCompleted := THIS^.M_CompleteStations();
END_IF
END_METHOD

(* This state should safely pause task executions without completely ending or
resetting them. *)
METHOD M401_Holding : BOOL
VAR_OUTPUT
	(* This should be set to true once all execution tasks are safely paused.
	Once set to true, the state machine will move to the 'Held' state. *)
	bHeld	: BOOL;
	(* This should be set to true if an external source requests that the module
	exit its current state and come to a controlled stop. Once set to true, the
	state machine will move to the 'Stopping' state. *)
	bStop	: BOOL;
	(* This should be set to true if a potentially hazardous error or a safety
	fault has occurred in any tasks. Once set to true, the state machine will
	move to the 'Aborting' state. *)
	bAbort	: BOOL;
END_VAR
IF THIS^.P_bError THEN
	bAbort := TRUE;
ELSE
	bHeld := THIS^.M_HoldStations();
END_IF
END_METHOD

(* In this state, the module and its components should be returned to the
scenario it was in before it entered the 'Holding' step so that the
'Execute' state can pick up where it left off. *)
METHOD M421_Unholding : BOOL
VAR_OUTPUT
	(* This should be set to true once the module is ready to restart
	execution. Once set to true, the state machine will move to the 'Execute'
	state. *)
	bUnheld	: BOOL;
	(* This should be set to true if an external source requests that the module
	exit its current state and come to a controlled stop. Once set to true, the
	state machine will move to the 'Stopping' state. *)
	bStop	: BOOL;
	(* This should be set to true if a potentially hazardous error or a safety
	fault has occurred in any tasks. Once set to true, the state machine will
	move to the 'Aborting' state. *)
	bAbort	: BOOL;
END_VAR
IF THIS^.P_bError THEN
	bAbort := TRUE;
ELSE
	bUnheld := THIS^.M_UnholdStations();
END_IF
END_METHOD

(* This state should safely pause task executions without completely ending or
resetting them. *)
METHOD M501_Suspending : BOOL
VAR_OUTPUT
	(* This should be set to true once all execution tasks are safely paused.
	Once set to true, the state machine will move to the 'Suspended' state. *)
	bSuspended	: BOOL;
	(* This should be set to true if an external source requests that the module
	exit its current state and come to a controlled stop. Once set to true, the
	state machine will move to the 'Stopping' state. *)
	bStop	: BOOL;
	(* This should be set to true if a potentially hazardous error or a safety
	fault has occurred in any tasks. Once set to true, the state machine will
	move to the 'Aborting' state. *)
	bAbort	: BOOL;
END_VAR
IF THIS^.P_bError THEN
	bAbort := TRUE;
ELSE
	bSuspended := THIS^.M_SuspendStations();
END_IF
END_METHOD

(* In this state, the module and its components should be returned to the
scenario it was in before it entered the 'Suspending' step so that the
'Execute' state can pick up where it left off. *)
METHOD M521_Unsuspending : BOOL
VAR_OUTPUT
	(* This should be set to true once the module is ready to restart
	execution. Once set to true, the state machine will move to the 'Execute'
	state. *)
	bUnsuspended	: BOOL;
	(* This should be set to true if an external source requests that the module
	exit its current state and come to a controlled stop. Once set to true, the
	state machine will move to the 'Stopping' state. *)
	bStop	: BOOL;
	(* This should be set to true if a potentially hazardous error or a safety
	fault has occurred in any tasks. Once set to true, the state machine will
	move to the 'Aborting' state. *)
	bAbort	: BOOL;
END_VAR
IF THIS^.P_bError THEN
	bAbort := TRUE;
ELSE
	bUnsuspended := THIS^.M_UnsuspendStations();
END_IF
END_METHOD

(* Executes M_Abort on all stations and returns TRUE when M_Abort
	returns TRUE on all stations. *)
METHOD M_AbortStations : BOOL
VAR CONSTANT
	_udintERROR_CODE: UDINT := E_MachineError.StationError;
	_strERROR_MSG: T_MaxString := 'A station had an error while trying to complete!';
END_VAR
VAR_INST
	_inst_arrResults : ARRAY[1..GVL_Constants.uintMAX_MACHINE_STATION_COUNT] OF BOOL;
END_VAR
VAR
	_intStep : INT;
	_uintIndex : UINT;
	_bResult : BOOL;
	_bComplete: BOOL;
END_VAR
_bResult := FALSE;
_intStep := mac_intAbortStationsStep;
CASE _intStep OF
	0: // Reset the results array
		M_ResetCommands();
		FOR _uintIndex := 1 TO GVL_Constants.uintMAX_MACHINE_STATION_COUNT DO
			_inst_arrResults[_uintIndex] := FALSE;
		END_FOR
		_intStep := _intStep + 10;
				
	10: // Call the method on each station
		_bComplete := TRUE;
		FOR _uintIndex := 1 TO GVL_Constants.uintMAX_MACHINE_STATION_COUNT DO
			
			// If the method hasn't finished for this device yet, call it
			IF mac_arrStations[_uintIndex] > 0 AND NOT _inst_arrResults[_uintIndex] THEN
				
				// Call the method
				_inst_arrResults[_uintIndex] := mac_arrStations[_uintIndex]^.M_Abort();
				
				// If the method did not complete, set complete to false
				IF NOT _inst_arrResults[_uintIndex] THEN
					_bComplete := FALSE;
				END_IF
			END_IF
		END_FOR
		
		// If all methods were successful, go to the next step
		IF _bComplete THEN
			_intStep := _intStep + 10;
		END_IF
		
	20: // Return TRUE and reset
		_bResult := TRUE;
		_intStep := 0;
END_CASE
mac_intAbortStationsStep := _intStep;
M_AbortStations := _bResult;
END_METHOD

(* Executes M_Clear on all stations and returns TRUE when M_Clear
	returns TRUE on all stations. *)
METHOD M_ClearStations : BOOL
VAR CONSTANT
	_udintERROR_CODE: UDINT := E_MachineError.StationError;
	_strERROR_MSG: T_MaxString := 'A station had an error while trying to clear!';
END_VAR
VAR_INST
	_inst_arrResults : ARRAY[1..GVL_Constants.uintMAX_MACHINE_STATION_COUNT] OF BOOL;
END_VAR
VAR
	_intStep : INT;
	_uintIndex : UINT;
	_bResult : BOOL;
	_bComplete: BOOL;
END_VAR
_bResult := FALSE;
_intStep := mac_intClearStationsStep;
CASE _intStep OF
	0: // Reset the results array
		M_ResetCommands();
		IF NOT THIS^.P_bError THEN
			FOR _uintIndex := 1 TO GVL_Constants.uintMAX_MACHINE_STATION_COUNT DO
				_inst_arrResults[_uintIndex] := FALSE;
			END_FOR
			_intStep := _intStep + 10;
		END_IF
	
	10: // Clear the errors on all stations
		FOR _uintIndex := 1 TO GVL_Constants.uintMAX_MACHINE_STATION_COUNT DO
			IF mac_arrStations[_uintIndex] > 0 AND NOT _inst_arrResults[_uintIndex] THEN
				mac_arrStations[_uintIndex]^.M_ClearError();
			END_IF
		END_FOR
		_intStep := _intStep + 10;
				
	20: // Call the method on each station
		_bComplete := TRUE;
		FOR _uintIndex := 1 TO GVL_Constants.uintMAX_MACHINE_STATION_COUNT DO
			
			// If the method hasn't finished for this device yet, call it
			IF mac_arrStations[_uintIndex] > 0 AND NOT _inst_arrResults[_uintIndex] THEN
				
				// Call the method
				_inst_arrResults[_uintIndex] := mac_arrStations[_uintIndex]^.M_Clear();
				
				// If there is an error, elevate it
				IF mac_arrStations[_uintIndex]^.P_bError THEN
					_bComplete := FALSE;
					THIS^.M_SetError(_udintERROR_CODE, _strERROR_MSG);
					_intStep := 0;
					
				// If the method did not complete, set complete to false
				ELSIF NOT _inst_arrResults[_uintIndex] THEN
					_bComplete := FALSE;
					
				END_IF
			END_IF
		END_FOR
		
		// If all methods were successful, go to the next step
		IF _bComplete THEN
			_intStep := _intStep + 10;
		END_IF
		
	30: // Return TRUE and reset
		_bResult := TRUE;
		_intStep := 0;
END_CASE
mac_intClearStationsStep := _intStep;
M_ClearStations := _bResult;
END_METHOD

(* Executes M_Complete on all stations and returns TRUE when M_Complete
	returns TRUE on all stations. *)
METHOD M_CompleteStations : BOOL
VAR CONSTANT
	_udintERROR_CODE: UDINT := E_MachineError.StationError;
	_strERROR_MSG: T_MaxString := 'A station had an error while trying to complete!';
END_VAR
VAR_INST
	_inst_arrResults : ARRAY[1..GVL_Constants.uintMAX_MACHINE_STATION_COUNT] OF BOOL;
END_VAR
VAR
	_intStep : INT;
	_uintIndex : UINT;
	_bResult : BOOL;
	_bComplete: BOOL;
END_VAR
_bResult := FALSE;
_intStep := mac_intCompleteStationsStep;
CASE _intStep OF
	0: // Reset the results array
		M_ResetCommands();
		IF NOT THIS^.P_bError THEN
			FOR _uintIndex := 1 TO GVL_Constants.uintMAX_MACHINE_STATION_COUNT DO
				_inst_arrResults[_uintIndex] := FALSE;
			END_FOR
			_intStep := _intStep + 10;
		END_IF
				
	10: // Call the method on each station
		_bComplete := TRUE;
		FOR _uintIndex := 1 TO GVL_Constants.uintMAX_MACHINE_STATION_COUNT DO
			
			// If the method hasn't finished for this device yet, call it
			IF mac_arrStations[_uintIndex] > 0 AND NOT _inst_arrResults[_uintIndex] THEN
				
				// Call the method
				_inst_arrResults[_uintIndex] := mac_arrStations[_uintIndex]^.M_Complete();
				
				// If there is an error, elevate it
				IF mac_arrStations[_uintIndex]^.P_bError THEN
					_bComplete := FALSE;
					THIS^.M_SetError(_udintERROR_CODE, _strERROR_MSG);
					_intStep := 0;
					
				// If the method did not complete, set complete to false
				ELSIF NOT _inst_arrResults[_uintIndex] THEN
					_bComplete := FALSE;
				END_IF
			END_IF
		END_FOR
		
		// If all methods were successful, go to the next step
		IF _bComplete THEN
			_intStep := _intStep + 10;
		END_IF
		
	20: // Return TRUE and reset
		_bResult := TRUE;
		_intStep := 0;
END_CASE
mac_intCompleteStationsStep := _intStep;
M_CompleteStations := _bResult;
END_METHOD

(* Executes M_Hold on all stations and returns TRUE when M_Hold 
	returns TRUE on all stations. *)
METHOD M_HoldStations : BOOL
VAR CONSTANT
	_udintERROR_CODE: UDINT := E_MachineError.StationError;
	_strERROR_MSG: T_MaxString := 'A station had an error while trying to complete!';
END_VAR
VAR_INST
	_inst_arrResults : ARRAY[1..GVL_Constants.uintMAX_MACHINE_STATION_COUNT] OF BOOL;
END_VAR
VAR
	_intStep : INT;
	_uintIndex : UINT;
	_bResult : BOOL;
	_bComplete: BOOL;
END_VAR
_bResult := FALSE;
_intStep := mac_intHoldStationsStep;
CASE _intStep OF
	0: // Reset the results array
		M_ResetCommands();
		IF NOT THIS^.P_bError THEN
			FOR _uintIndex := 1 TO GVL_Constants.uintMAX_MACHINE_STATION_COUNT DO
				_inst_arrResults[_uintIndex] := FALSE;
			END_FOR
			_intStep := _intStep + 10;
		END_IF
				
	10: // Call the method on each station
		_bComplete := TRUE;
		FOR _uintIndex := 1 TO GVL_Constants.uintMAX_MACHINE_STATION_COUNT DO
			
			// If the method hasn't finished for this device yet, call it
			IF mac_arrStations[_uintIndex] > 0 AND NOT _inst_arrResults[_uintIndex] THEN
				
				// Call the method
				_inst_arrResults[_uintIndex] := mac_arrStations[_uintIndex]^.M_Hold();
				
				// If there is an error, elevate it
				IF mac_arrStations[_uintIndex]^.P_bError THEN
					_bComplete := FALSE;
					THIS^.M_SetError(_udintERROR_CODE, _strERROR_MSG);
					_intStep := 0;
					
				// If the method did not complete, set complete to false
				ELSIF NOT _inst_arrResults[_uintIndex] THEN
					_bComplete := FALSE;
				END_IF
			END_IF
		END_FOR
		
		// If all methods were successful, go to the next step
		IF _bComplete THEN
			_intStep := _intStep + 10;
		END_IF
		
	20: // Return TRUE and reset
		_bResult := TRUE;
		_intStep := 0;
END_CASE
mac_intHoldStationsStep := _intStep;
M_HoldStations := _bResult;
END_METHOD

(* Executes M_Reset on all stations and returns TRUE when M_Reset 
	returns TRUE on all stations. *)
METHOD M_ResetStations : BOOL
VAR CONSTANT
	_udintERROR_CODE: UDINT := E_MachineError.StationError;
	_strERROR_MSG: T_MaxString := 'A station had an error while trying to complete!';
END_VAR
VAR_INST
	_inst_arrResults : ARRAY[1..GVL_Constants.uintMAX_MACHINE_STATION_COUNT] OF BOOL;
END_VAR
VAR
	_intStep : INT;
	_uintIndex : UINT;
	_bResult : BOOL;
	_bComplete: BOOL;
END_VAR
_bResult := FALSE;
_intStep := mac_intResetStationsStep;
CASE _intStep OF
	0: // Reset the results array
		M_ResetCommands();
		IF NOT THIS^.P_bError THEN
			FOR _uintIndex := 1 TO GVL_Constants.uintMAX_MACHINE_STATION_COUNT DO
				_inst_arrResults[_uintIndex] := FALSE;
			END_FOR
			_intStep := _intStep + 10;
		END_IF
				
	10: // Call the method on each station
		_bComplete := TRUE;
		FOR _uintIndex := 1 TO GVL_Constants.uintMAX_MACHINE_STATION_COUNT DO
			
			// If the method hasn't finished for this device yet, call it
			IF mac_arrStations[_uintIndex] > 0 AND NOT _inst_arrResults[_uintIndex] THEN
				
				// Call the method
				_inst_arrResults[_uintIndex] := mac_arrStations[_uintIndex]^.M_Reset();
				
				// If there is an error, elevate it
				IF mac_arrStations[_uintIndex]^.P_bError THEN
					_bComplete := FALSE;
					THIS^.M_SetError(_udintERROR_CODE, _strERROR_MSG);
					_intStep := 0;
					
				// If the method did not complete, set complete to false
				ELSIF NOT _inst_arrResults[_uintIndex] THEN
					_bComplete := FALSE;
				END_IF
			END_IF
		END_FOR
		
		// If all methods were successful, go to the next step
		IF _bComplete THEN
			_intStep := _intStep + 10;
		END_IF
		
	20: // Return TRUE and reset
		_bResult := TRUE;
		_intStep := 0;
END_CASE
mac_intResetStationsStep := _intStep;
M_ResetStations := _bResult;
END_METHOD

(* Executes M_Start on all stations and returns TRUE when M_Start 
	returns TRUE on all stations. *)
METHOD M_StartStations : BOOL
VAR CONSTANT
	_udintERROR_CODE: UDINT := E_MachineError.StationError;
	_strERROR_MSG: T_MaxString := 'A station had an error while trying to complete!';
END_VAR
VAR_INST
	_inst_arrResults : ARRAY[1..GVL_Constants.uintMAX_MACHINE_STATION_COUNT] OF BOOL;
END_VAR
VAR
	_intStep : INT;
	_uintIndex : UINT;
	_bResult : BOOL;
	_bComplete: BOOL;
END_VAR
_bResult := FALSE;
_intStep := mac_intStartStationsStep;
CASE _intStep OF
	0: // Reset the results array
		M_ResetCommands();
		IF NOT THIS^.P_bError THEN
			FOR _uintIndex := 1 TO GVL_Constants.uintMAX_MACHINE_STATION_COUNT DO
				_inst_arrResults[_uintIndex] := FALSE;
			END_FOR
			_intStep := _intStep + 10;
		END_IF
				
	10: // Call the method on each station
		_bComplete := TRUE;
		FOR _uintIndex := 1 TO GVL_Constants.uintMAX_MACHINE_STATION_COUNT DO
			
			// If the method hasn't finished for this device yet, call it
			IF mac_arrStations[_uintIndex] > 0 AND NOT _inst_arrResults[_uintIndex] THEN
				
				// Call the method
				_inst_arrResults[_uintIndex] := mac_arrStations[_uintIndex]^.M_Start();
				
				// If there is an error, elevate it
				IF mac_arrStations[_uintIndex]^.P_bError THEN
					_bComplete := FALSE;
					THIS^.M_SetError(_udintERROR_CODE, _strERROR_MSG);
					_intStep := 0;
					
				// If the method did not complete, set complete to false
				ELSIF NOT _inst_arrResults[_uintIndex] THEN
					_bComplete := FALSE;
				END_IF
			END_IF
		END_FOR
		
		// If all methods were successful, go to the next step
		IF _bComplete THEN
			_intStep := _intStep + 10;
		END_IF
		
	20: // Return TRUE and reset
		_bResult := TRUE;
		_intStep := 0;
END_CASE
mac_intStartStationsStep := _intStep;
M_StartStations := _bResult;
END_METHOD

(* Executes M_Stop on all stations and returns TRUE when M_Stop 
	returns TRUE on all stations. *)
METHOD M_StopStations : BOOL
VAR CONSTANT
	_udintERROR_CODE: UDINT := E_MachineError.StationError;
	_strERROR_MSG: T_MaxString := 'A station had an error while trying to complete!';
END_VAR
VAR_INST
	_inst_arrResults : ARRAY[1..GVL_Constants.uintMAX_MACHINE_STATION_COUNT] OF BOOL;
END_VAR
VAR
	_intStep : INT;
	_uintIndex : UINT;
	_bResult : BOOL;
	_bComplete: BOOL;
END_VAR
_bResult := FALSE;
_intStep := mac_intStopStationsStep;
CASE _intStep OF
	0: // Reset the results array
		M_ResetCommands();
		IF NOT THIS^.P_bError THEN
			FOR _uintIndex := 1 TO GVL_Constants.uintMAX_MACHINE_STATION_COUNT DO
				_inst_arrResults[_uintIndex] := FALSE;
			END_FOR
			_intStep := _intStep + 10;
		END_IF
				
	10: // Call the method on each station
		_bComplete := TRUE;
		FOR _uintIndex := 1 TO GVL_Constants.uintMAX_MACHINE_STATION_COUNT DO
			
			// If the method hasn't finished for this device yet, call it
			IF mac_arrStations[_uintIndex] > 0 AND NOT _inst_arrResults[_uintIndex] THEN
				
				// Call the method
				_inst_arrResults[_uintIndex] := mac_arrStations[_uintIndex]^.M_Stop();
				
				// If there is an error, elevate it
				IF mac_arrStations[_uintIndex]^.P_bError THEN
					_bComplete := FALSE;
					THIS^.M_SetError(_udintERROR_CODE, _strERROR_MSG);
					_intStep := 0;
					
				// If the method did not complete, set complete to false
				ELSIF NOT _inst_arrResults[_uintIndex] THEN
					_bComplete := FALSE;
				END_IF
			END_IF
		END_FOR
		
		// If all methods were successful, go to the next step
		IF _bComplete THEN
			_intStep := _intStep + 10;
		END_IF
		
	20: // Return TRUE and reset
		_bResult := TRUE;
		_intStep := 0;
END_CASE
mac_intStopStationsStep := _intStep;
M_StopStations := _bResult;
END_METHOD

(* Executes M_Suspend on all stations and returns TRUE when M_Suspend
	returns TRUE on all stations. *)
METHOD M_SuspendStations : BOOL
VAR CONSTANT
	_udintERROR_CODE: UDINT := E_MachineError.StationError;
	_strERROR_MSG: T_MaxString := 'A station had an error while trying to complete!';
END_VAR
VAR_INST
	_inst_arrResults : ARRAY[1..GVL_Constants.uintMAX_MACHINE_STATION_COUNT] OF BOOL;
END_VAR
VAR
	_intStep : INT;
	_uintIndex : UINT;
	_bResult : BOOL;
	_bComplete: BOOL;
END_VAR
_bResult := FALSE;
_intStep := mac_intSuspendStationsStep;
CASE _intStep OF
	0: // Reset the results array
		M_ResetCommands();
		IF NOT THIS^.P_bError THEN
			FOR _uintIndex := 1 TO GVL_Constants.uintMAX_MACHINE_STATION_COUNT DO
				_inst_arrResults[_uintIndex] := FALSE;
			END_FOR
			_intStep := _intStep + 10;
		END_IF
				
	10: // Call the method on each station
		_bComplete := TRUE;
		FOR _uintIndex := 1 TO GVL_Constants.uintMAX_MACHINE_STATION_COUNT DO
			
			// If the method hasn't finished for this device yet, call it
			IF mac_arrStations[_uintIndex] > 0 AND NOT _inst_arrResults[_uintIndex] THEN
				
				// Call the method
				_inst_arrResults[_uintIndex] := mac_arrStations[_uintIndex]^.M_Suspend();
				
				// If there is an error, elevate it
				IF mac_arrStations[_uintIndex]^.P_bError THEN
					_bComplete := FALSE;
					THIS^.M_SetError(_udintERROR_CODE, _strERROR_MSG);
					_intStep := 0;
					
				// If the method did not complete, set complete to false
				ELSIF NOT _inst_arrResults[_uintIndex] THEN
					_bComplete := FALSE;
				END_IF
			END_IF
		END_FOR
		
		// If all methods were successful, go to the next step
		IF _bComplete THEN
			_intStep := _intStep + 10;
		END_IF
		
	20: // Return TRUE and reset
		_bResult := TRUE;
		_intStep := 0;
END_CASE
mac_intSuspendStationsStep := _intStep;
M_SuspendStations := _bResult;
END_METHOD

(* Executes M_Unhold on all stations and returns TRUE when M_Unhold
	returns TRUE on all stations. *)
METHOD M_UnholdStations : BOOL
VAR CONSTANT
	_udintERROR_CODE: UDINT := E_MachineError.StationError;
	_strERROR_MSG: T_MaxString := 'A station had an error while trying to complete!';
END_VAR
VAR_INST
	_inst_arrResults : ARRAY[1..GVL_Constants.uintMAX_MACHINE_STATION_COUNT] OF BOOL;
END_VAR
VAR
	_intStep : INT;
	_uintIndex : UINT;
	_bResult : BOOL;
	_bComplete: BOOL;
END_VAR
_bResult := FALSE;
_intStep := mac_intUnholdStationsStep;
CASE _intStep OF
	0: // Reset the results array
		M_ResetCommands();
		IF NOT THIS^.P_bError THEN
			FOR _uintIndex := 1 TO GVL_Constants.uintMAX_MACHINE_STATION_COUNT DO
				_inst_arrResults[_uintIndex] := FALSE;
			END_FOR
			_intStep := _intStep + 10;
		END_IF
				
	10: // Call the method on each station
		_bComplete := TRUE;
		FOR _uintIndex := 1 TO GVL_Constants.uintMAX_MACHINE_STATION_COUNT DO
			
			// If the method hasn't finished for this device yet, call it
			IF mac_arrStations[_uintIndex] > 0 AND NOT _inst_arrResults[_uintIndex] THEN
				
				// Call the method
				_inst_arrResults[_uintIndex] := mac_arrStations[_uintIndex]^.M_Unhold();
				
				// If there is an error, elevate it
				IF mac_arrStations[_uintIndex]^.P_bError THEN
					_bComplete := FALSE;
					THIS^.M_SetError(_udintERROR_CODE, _strERROR_MSG);
					_intStep := 0;
					
				// If the method did not complete, set complete to false
				ELSIF NOT _inst_arrResults[_uintIndex] THEN
					_bComplete := FALSE;
				END_IF
			END_IF
		END_FOR
		
		// If all methods were successful, go to the next step
		IF _bComplete THEN
			_intStep := _intStep + 10;
		END_IF
		
	20: // Return TRUE and reset
		_bResult := TRUE;
		_intStep := 0;
END_CASE
mac_intUnholdStationsStep := _intStep;
M_UnholdStations := _bResult;
END_METHOD

(* Executes M_Unsuspend on all stations and returns TRUE when M_Unsuspend
	returns TRUE on all stations. *)
METHOD M_UnsuspendStations : BOOL
VAR CONSTANT
	_udintERROR_CODE: UDINT := E_MachineError.StationError;
	_strERROR_MSG: T_MaxString := 'A station had an error while trying to complete!';
END_VAR
VAR_INST
	_inst_arrResults : ARRAY[1..GVL_Constants.uintMAX_MACHINE_STATION_COUNT] OF BOOL;
END_VAR
VAR
	_intStep : INT;
	_uintIndex : UINT;
	_bResult : BOOL;
	_bComplete: BOOL;
END_VAR
_bResult := FALSE;
_intStep := mac_intUnsuspendStationsStep;
CASE _intStep OF
	0: // Reset the results array
		M_ResetCommands();
		IF NOT THIS^.P_bError THEN
			FOR _uintIndex := 1 TO GVL_Constants.uintMAX_MACHINE_STATION_COUNT DO
				_inst_arrResults[_uintIndex] := FALSE;
			END_FOR
			_intStep := _intStep + 10;
		END_IF
				
	10: // Call the method on each station
		_bComplete := TRUE;
		FOR _uintIndex := 1 TO GVL_Constants.uintMAX_MACHINE_STATION_COUNT DO
			
			// If the method hasn't finished for this device yet, call it
			IF mac_arrStations[_uintIndex] > 0 AND NOT _inst_arrResults[_uintIndex] THEN
				
				// Call the method
				_inst_arrResults[_uintIndex] := mac_arrStations[_uintIndex]^.M_Unsuspend();
				
				// If there is an error, elevate it
				IF mac_arrStations[_uintIndex]^.P_bError THEN
					_bComplete := FALSE;
					THIS^.M_SetError(_udintERROR_CODE, _strERROR_MSG);
					_intStep := 0;
					
				// If the method did not complete, set complete to false
				ELSIF NOT _inst_arrResults[_uintIndex] THEN
					_bComplete := FALSE;
				END_IF
			END_IF
		END_FOR
		
		// If all methods were successful, go to the next step
		IF _bComplete THEN
			_intStep := _intStep + 10;
		END_IF
		
	20: // Return TRUE and reset
		_bResult := TRUE;
		_intStep := 0;
END_CASE
mac_intUnsuspendStationsStep := _intStep;
M_UnsuspendStations := _bResult;
END_METHOD

(* Check all stations in the station list for errors and
	raise an error if there is one. *)
METHOD M_CheckStations : BOOL

VAR
	_uintIndex: UINT;
	_fbStation: POINTER TO FB_Station;
	_udintErrorNo: UDINT;
	_strErrorDescription: T_MaxString;
END_VAR
M_CheckStations := FALSE;
// Run through each device
FOR _uintIndex := 1 TO GVL_Constants.uintMAX_MACHINE_STATION_COUNT DO
	// If the pointer is set
	IF mac_arrStations[_uintIndex] > 0 THEN
		// Get the device from the pointer
		_fbStation := mac_arrStations[_uintIndex];
		
		// Check device for error and set error if there is one
		IF _fbStation^.P_bError THEN
			_udintErrorNo := E_MachineError.StationError;
			_udintErrorNo := _udintErrorNo + _uintIndex;
			_strErrorDescription := CONCAT('Station ', _fbStation^.in_strUniqueId);
			_strErrorDescription := CONCAT(_strErrorDescription, ' has the following error: (');
			_strErrorDescription := CONCAT(_strErrorDescription, UDINT_TO_STRING(_fbStation^.P_udintErrorCode));
			_strErrorDescription := CONCAT(_strErrorDescription, ') ');
			_strErrorDescription := CONCAT(_strErrorDescription, _fbStation^.P_strErrorMessage);
			
			THIS^.M_SetError(
				_udintErrorNo,
				_strErrorDescription);
				
			M_CheckStations := TRUE;
		END_IF
	END_IF
END_FOR
END_METHOD

{attribute 'hide'}
(* Adds a station to the station list. *)
METHOD PROTECTED M_SetStation : BOOL
VAR_INPUT
	(* Index of station to set. Between 1 and uintMAX_MACHINE_STATION_COUNT. *)
	uintIndex: UINT;
	
	(* Reference to the station to be set in the station list. *)
	refStation: REFERENCE TO FB_Station;
END_VAR
IF __ISVALIDREF(refStation) AND uintIndex > 0 AND uintIndex <= GVL_Constants.uintMAX_STATION_DEVICE_COUNT THEN
	mac_arrStations[uintIndex] := ADR(refStation);
	M_SetStation := TRUE;
ELSE
	M_SetStation := FALSE;
END_IF
END_METHOD

(* The array of station pointers for this machine. *)
PROPERTY P_arrStations : T_MachineStationArray
GET
P_arrStations := mac_arrStations;
END_GET
END_PROPERTY

END_FUNCTION_BLOCK

// Interfaces/State Machine/Stateful/I_Stateful
(* The stateful interface implements a full PackML state machine, including
the entry and exit methods. Implement I_SimpleStateful instead if you are not
planning to use entry and exit methods. *)
INTERFACE I_Stateful EXTENDS I_WaitingStatesOnly, I_TransitionStatesOnly

END_INTERFACE

// Interfaces/State Machine/Stateful/I_SimpleStateful
(* The simple stateful interface implements only the "DO" portions of the
PackML states. The ENTRY and EXIT methods are not included. *)
INTERFACE I_SimpleStateful EXTENDS I_SimpleWaitingStatesOnly, I_SimpleTransitionStatesOnly

END_INTERFACE

// Interfaces/State Machine/Stateful/I_SimpleWaitingStatesOnly
(* This interface implements only the PackML waiting states. 
This only includes the DO methods (no ENTRY or EXIT). *)
INTERFACE I_SimpleWaitingStatesOnly EXTENDS I_SimpleExecuteStateOnly

(* This state is entered after the aborting state completes, and should
not modify anything in the module while awaiting an explicit 'Clear' command. *)
METHOD M011_Aborted : BOOL
VAR_INPUT
END_VAR
VAR_OUTPUT
	(* This should be set to true once an explicit 'Clear' command is received.
	Once set to true, the state machine will move to the 'Clearing' state. *)
	bClear : BOOL;
END_VAR
END_METHOD

(* The machine should be stationary and awaiting an explicit 'Reset' command
while in this state. Once the 'Reset' command is received, the state machine
will move to the 'Resetting' state. *)
METHOD M111_Stopped : BOOL
VAR_INPUT
END_VAR
VAR_OUTPUT
	(* This should be set to true if an explicit reset command is received.
	Once set to true, the state machine will move to the 'Resetting' state. *)
	bReset : BOOL;
	
	(* This should be set to true if a potentially hazardous error or a safety
	fault has occurred in any tasks. Once set to true, the state machine will
	move to the 'Aborting' state. *)
	bAbort : BOOL; 
END_VAR
END_METHOD

(* This state should maintain the status of the module and its components that
was set by the resetting step while awaiting an explicit 'Start' command. *)
METHOD M211_Idle : BOOL
VAR_INPUT
END_VAR
VAR_OUTPUT
	(* This should be set to true if an explicit 'Start' command is received.
	Once set to true, the state machine will move to the 'Starting' state. *)
	bStart : BOOL;
	
	(* This should be set to true if an external source requests that the module
	exit its current state and come to a controlled stop. Once set to true, the
	state machine will move to the 'Stopping' state. *)
	bStop : BOOL;
	
	(* This should be set to true if a potentially hazardous error or a safety
	fault has occurred in any tasks. Once set to true, the state machine will
	move to the 'Aborting' state. *)
	bAbort : BOOL;
END_VAR
END_METHOD

(* The module should remain stationary within this state while maintaing any
execution statistics and awaiting an explicit 'Return' command. *)
METHOD M331_Complete : BOOL
VAR_INPUT
END_VAR
VAR_OUTPUT
	(* This should be set to true if an explicit 'Return' command is received.
	Once set to true, the state machine will move to the 'Resetting' state. *)
	bReturn : BOOL;
	
	(* This should be set to true if an external source requests that the module
	exit its current state and come to a controlled stop. Once set to true, the
	state machine will move to the 'Stopping' state. *)
	bStop : BOOL;
	
	(* This should be set to true if a potentially hazardous error or a safety
	fault has occurred in any tasks. Once set to true, the state machine will
	move to the 'Aborting' state. *)
	bAbort : BOOL;
END_VAR
END_METHOD

(* In this state the most recent execution status should be maintained while
awaiting an explicit 'Unhold' command once internal conditions are satisfactory. *)
METHOD M411_Held : BOOL
VAR_INPUT
END_VAR
VAR_OUTPUT
	(* This should be set to true if an explicit 'Unhold' command is received.
	Once set to true, the state machine will move to the 'Unholding' state. *)
	bUnhold : BOOL;
	
	(* This should be set to true if an external source requests that the module
	exit its current state and come to a controlled stop. Once set to true, the
	state machine will move to the 'Stopping' state. *)
	bStop : BOOL;
	
	(* This should be set to true if a potentially hazardous error or a safety
	fault has occurred in any tasks. Once set to true, the state machine will
	move to the 'Aborting' state. *)
	bAbort : BOOL;
END_VAR
END_METHOD

(* In this state the most recent execution status should be maintained while
awaiting an explicit 'Unsuspend' command once external conditions are satisfactory. *)
METHOD M511_Suspended : BOOL
VAR_INPUT
END_VAR
VAR_OUTPUT
	(* This should be set to true if an explicit 'Unsuspend' command is received.
	Once set to true, the state machine will move to the 'Unsuspending' state. *)
	bUnsuspend : BOOL;
	
	(* This should be set to true if an external source requests that the module
	exit its current state and come to a controlled stop. Once set to true, the
	state machine will move to the 'Stopping' state. *)
	bStop : BOOL;
	
	(* This should be set to true if a potentially hazardous error or a safety
	fault has occurred in any tasks. Once set to true, the state machine will
	move to the 'Aborting' state. *)
	bAbort : BOOL;
END_VAR
END_METHOD

END_INTERFACE

// Interfaces/State Machine/Stateful/I_SimpleExecuteStateOnly
(* This interface only implements the methods for the Execute state.
Only includes the DO method, no ENTRY or EXIT. *)
INTERFACE I_SimpleExecuteStateOnly

(* The module should remain in this state while it is actively performing
automated tasks. Once all work is finished the state machine should move to the
'Completing' state. *)
METHOD M311_Execute : BOOL
VAR_INPUT
END_VAR
VAR_OUTPUT
	(* This should be set to true once all tasks are complete and automated
	execution should be ended. Once set to true, the state machine will move to
	the 'Completing' state. *)
	bFinished : BOOL;
	
	(* This should be set to true as a result of an explicit 'Hold' command
	or if internal conditions require the module to stop operation without
	completely exiting the execution sequence. Once set to true, the state
	machine will move to the 'Holding' state. *)
	bHold : BOOL;
	
	(* This should be set to true if external conditions require the module to
	suspend operation until the external conditions are cleared. Once set to
	true, the state machine will move to the 'Suspending' state. *)
	bSuspend : BOOL;
	
	(* This should be set to true if an external source requests that the module
	exit its current state and come to a controlled stop. Once set to true, the
	state machine will move to the 'Stopping' state. *)
	bStop : BOOL;
	
	(* This should be set to true if a potentially hazardous error or a safety
	fault has occurred in any tasks. Once set to true, the state machine will
	move to the 'Aborting' state. *)
	bAbort : BOOL;
END_VAR
END_METHOD

END_INTERFACE

// Interfaces/State Machine/Stateful/I_SimpleTransitionStatesOnly
(* This interface implements only the PackML transition states. 
This only includes the DO methods (no ENTRY or EXIT). *)
INTERFACE I_SimpleTransitionStatesOnly

(* The 'Aborting' state can be entered at any time while within the 'abortable'
section of the state machine. It is typically entered in response to an 'Abort'
command or a critical fault. The logic should safely but rapidly bring the
components of the module to a stop while maintaining as much information about
the pre-abort scenario as possible. *)
METHOD M001_Aborting : BOOL
VAR_INPUT
END_VAR
VAR_OUTPUT
	(* This should be set to true once all components of the module have safely
	come to a stop. Once set to true, the state machine will move to the
	'Aborted' state. *)
	bAborted : BOOL;
END_VAR
END_METHOD

(* This state should clear any faults and reset any safety features related
to the module, as well as perform actions similar to the 'Stopping' state
if they were not already performed while aborting. *)
METHOD M021_Clearing : BOOL
VAR_INPUT
END_VAR
VAR_OUTPUT
	(* This should be set to true once the safety state of all module
	components are reset and all errors are cleared. *)
	bCleared : BOOL;
	
	(* This should be set to true if a potentially hazardous error or a safety
	fault has occurred in any tasks. Once set to true, the state machine will
	move to the 'Aborting' state. *)
	bAbort : BOOL;
END_VAR
END_METHOD

(* This state can be entered from anywhere within the 'stoppable' group of
states. This state should safely bring the components of the module to a
controlled stop and then move to the 'Stopped' state once completed. *)
METHOD M101_Stopping : BOOL
VAR_INPUT
END_VAR
VAR_OUTPUT
	(* This should be set to true once all relevant components have come to a
	controlled stop. Once set to true, the state machine will move to the
	'Stopped' state. *)
	bStopped : BOOL;
	
	(* This should be set to true if a potentially hazardous error or a safety
	fault has occurred in any tasks. Once set to true, the state machine will
	move to the 'Aborting' state. *)
	bAbort : BOOL;
END_VAR
END_METHOD

(* This state should place the module and all of its components into a safe
energized idle state where it will wait for a start command. Once all tasks are
complete, it will move to the 'Idle' state. No external movement should occur
as a result of this state. *)
METHOD M201_Resetting : BOOL
VAR_INPUT
END_VAR
VAR_OUTPUT
	(* Set this to true once the module is energized and ready to start.
	Once set to true, the state machine will move to the 'Idle' state. *)
	bIdle : BOOL;
	
	(* This should be set to true if an external source requests that the module
	exit its current state and come to a controlled stop. Once set to true, the
	state machine will move to the 'Stopping' state. *)
	bStop : BOOL;
	
	(* This should be set to true if a potentially hazardous error or a safety
	fault has occurred in any tasks. Once set to true, the state machine will
	move to the 'Aborting' state. *)
	bAbort : BOOL;
END_VAR
END_METHOD

(* This state should make any final preparations needed for the 'Execute' state
prior to entering the 'Execute' state. *)
METHOD M301_Starting : BOOL
VAR_INPUT
END_VAR
VAR_OUTPUT
	(* This should be set to true once the module and its components are fully
	prepared for process execution. Once set to true, the state machine will
	move to the 'Execute' state. *)
	bStarted : BOOL;
	
	(* This should be set to true if an external source requests that the module
	exit its current state and come to a controlled stop. Once set to true, the
	state machine will move to the 'Stopping' state. *)
	bStop : BOOL;
	
	(* This should be set to true if a potentially hazardous error or a safety
	fault has occurred in any tasks. Once set to true, the state machine will
	move to the 'Aborting' state. *)
	bAbort : BOOL;
END_VAR
END_METHOD

(* This state will perform any post-execution tasks prior to moving to the
'Completed' state. *)
METHOD M321_Completing : BOOL
VAR_INPUT
END_VAR
VAR_OUTPUT
	(* This should be set to true once all post-execution tasks are complete.
	Once set to true, the state machine will move to the 'Complete' state. *)
	bCompleted : BOOL; // Move to the Complete state
	
	(* This should be set to true if an external source requests that the module
	exit its current state and come to a controlled stop. Once set to true, the
	state machine will move to the 'Stopping' state. *)
	bStop : BOOL;
	
	(* This should be set to true if a potentially hazardous error or a safety
	fault has occurred in any tasks. Once set to true, the state machine will
	move to the 'Aborting' state. *)
	bAbort : BOOL;
END_VAR
END_METHOD

(* This state should safely pause task executions without completely ending or
resetting them. *)
METHOD M401_Holding : BOOL
VAR_INPUT
END_VAR
VAR_OUTPUT
	(* This should be set to true once all execution tasks are safely paused.
	Once set to true, the state machine will move to the 'Held' state. *)
	bHeld : BOOL;
	
	(* This should be set to true if an external source requests that the module
	exit its current state and come to a controlled stop. Once set to true, the
	state machine will move to the 'Stopping' state. *)
	bStop : BOOL;
	
	(* This should be set to true if a potentially hazardous error or a safety
	fault has occurred in any tasks. Once set to true, the state machine will
	move to the 'Aborting' state. *)
	bAbort : BOOL;
END_VAR
END_METHOD

(* In this state, the module and its components should be returned to the
scenario it was in before it entered the 'Holding' step so that the
'Execute' state can pick up where it left off. *)
METHOD M421_Unholding : BOOL
VAR_INPUT
END_VAR
VAR_OUTPUT
	(* This should be set to true once the module is ready to restart
	execution. Once set to true, the state machine will move to the 'Execute'
	state. *)
	bUnheld : BOOL;
	
	(* This should be set to true if an external source requests that the module
	exit its current state and come to a controlled stop. Once set to true, the
	state machine will move to the 'Stopping' state. *)
	bStop : BOOL;
	
	(* This should be set to true if a potentially hazardous error or a safety
	fault has occurred in any tasks. Once set to true, the state machine will
	move to the 'Aborting' state. *)
	bAbort : BOOL;
END_VAR
END_METHOD

(* This state should safely pause task executions without completely ending or
resetting them. *)
METHOD M501_Suspending : BOOL
VAR_INPUT
END_VAR
VAR_OUTPUT
	(* This should be set to true once all execution tasks are safely paused.
	Once set to true, the state machine will move to the 'Suspended' state. *)
	bSuspended : BOOL;
	
	(* This should be set to true if an external source requests that the module
	exit its current state and come to a controlled stop. Once set to true, the
	state machine will move to the 'Stopping' state. *)
	bStop : BOOL;
	
	(* This should be set to true if a potentially hazardous error or a safety
	fault has occurred in any tasks. Once set to true, the state machine will
	move to the 'Aborting' state. *)
	bAbort : BOOL;
END_VAR
END_METHOD

(* In this state, the module and its components should be returned to the
scenario it was in before it entered the 'Suspending' step so that the
'Execute' state can pick up where it left off. *)
METHOD M521_Unsuspending : BOOL
VAR_INPUT
END_VAR
VAR_OUTPUT
	(* This should be set to true once the module is ready to restart
	execution. Once set to true, the state machine will move to the 'Execute'
	state. *)
	bUnsuspended : BOOL;
	
	(* This should be set to true if an external source requests that the module
	exit its current state and come to a controlled stop. Once set to true, the
	state machine will move to the 'Stopping' state. *)
	bStop : BOOL;
	
	(* This should be set to true if a potentially hazardous error or a safety
	fault has occurred in any tasks. Once set to true, the state machine will
	move to the 'Aborting' state. *)
	bAbort : BOOL;
END_VAR
END_METHOD

END_INTERFACE

// Interfaces/State Machine/Stateful/I_WaitingStatesOnly
(* This interface implements only the PackML waiting states. *)
INTERFACE I_WaitingStatesOnly EXTENDS I_SimpleWaitingStatesOnly

(* Runs for a single cycle when entering the aborted state. *)
METHOD M010_Aborted_Entry : BOOL
VAR_INPUT
END_VAR
END_METHOD

(* Runs for a single cycle when exiting the aborted state. *)
METHOD M012_Aborted_Exit : BOOL
VAR_INPUT
END_VAR
END_METHOD

(* Runs for a single cycle when entering the stopped state. *)
METHOD M110_Stopped_Entry : BOOL
VAR_INPUT
END_VAR
END_METHOD

(* Runs for a single cycle when exiting the stopped state. *)
METHOD M112_Stopped_Exit : BOOL
VAR_INPUT
END_VAR
END_METHOD

(* Runs for a single cycle when entering the idle state. *)
METHOD M210_Idle_Entry : BOOL
VAR_INPUT
END_VAR
END_METHOD

(* Runs for a single cycle when exiting the idle state. *)
METHOD M212_Idle_Exit : BOOL
VAR_INPUT
END_VAR
END_METHOD

(* Runs for a single cycle when entering the execute state. *)
METHOD M310_Execute_Entry : BOOL
VAR_INPUT
END_VAR
END_METHOD

(* Runs for a single cycle when exiting the execute state. *)
METHOD M312_Execute_Exit : BOOL
VAR_INPUT
END_VAR
END_METHOD

(* Runs for a single cycle when entering the complete state. *)
METHOD M330_Complete_Entry : BOOL
VAR_INPUT
END_VAR
END_METHOD

(* Runs for a single cycle when exiting the complete state. *)
METHOD M332_Complete_Exit : BOOL
VAR_INPUT
END_VAR
END_METHOD

(* Runs for a single cycle when entering the held state. *)
METHOD M410_Held_Entry : BOOL
VAR_INPUT
END_VAR
END_METHOD

(* Runs for a single cycle when exiting the held state. *)
METHOD M412_Held_Exit : BOOL
VAR_INPUT
END_VAR
END_METHOD

(* Runs for a single cycle when entering the suspended state. *)
METHOD M510_Suspended_Entry : BOOL
VAR_INPUT
END_VAR
END_METHOD

(* Runs for a single cycle when exiting the suspended state. *)
METHOD M512_Suspended_Exit : BOOL
VAR_INPUT
END_VAR
END_METHOD

END_INTERFACE

// Interfaces/State Machine/Stateful/I_TransitionStatesOnly
(* This interface implements only the PackML transition states. *)
INTERFACE I_TransitionStatesOnly EXTENDS I_SimpleTransitionStatesOnly

(* Runs for a single cycle when entering the aborting state. *)
METHOD M000_Aborting_Entry : BOOL
VAR_INPUT
END_VAR
END_METHOD

(* Runs for a single cycle when exiting the aborting state. *)
METHOD M002_Aborting_Exit : BOOL
VAR_INPUT
END_VAR
END_METHOD

(* Runs for a single cycle when entering the clearing state. *)
METHOD M020_Clearing_Entry : BOOL
VAR_INPUT
END_VAR
END_METHOD

(* Runs for a single cycle when exiting the clearing state. *)
METHOD M022_Clearing_Exit : BOOL
VAR_INPUT
END_VAR
END_METHOD

(* Runs for a single cycle when entering the stopping state. *)
METHOD M100_Stopping_Entry : BOOL
VAR_INPUT
END_VAR
END_METHOD

(* Runs for a single cycle when exiting the stopping state. *)
METHOD M102_Stopping_Exit : BOOL
VAR_INPUT
END_VAR
END_METHOD

(* Runs for a single cycle when entering the resetting state. *)
METHOD M200_Resetting_Entry : BOOL
VAR_INPUT
END_VAR
END_METHOD

(* Runs for a single cycle when exiting the resetting state. *)
METHOD M202_Resetting_Exit : BOOL
VAR_INPUT
END_VAR
END_METHOD

(* Runs for a single cycle when entering the starting state. *)
METHOD M300_Starting_Entry : BOOL
VAR_INPUT
END_VAR
END_METHOD

(* Runs for a single cycle when exiting the starting state. *)
METHOD M302_Starting_Exit : BOOL
VAR_INPUT
END_VAR
END_METHOD

(* Runs for a single cycle when entering the completing state. *)
METHOD M320_Completing_Entry : BOOL
VAR_INPUT
END_VAR
END_METHOD

(* Runs for a single cycle when exiting the completing state. *)
METHOD M322_Completing_Exit : BOOL
VAR_INPUT
END_VAR
END_METHOD

(* Runs for a single cycle when entering the holding state. *)
METHOD M400_Holding_Entry : BOOL
VAR_INPUT
END_VAR
END_METHOD

(* Runs for a single cycle when exiting the holding state. *)
METHOD M402_Holding_Exit : BOOL
VAR_INPUT
END_VAR
END_METHOD

(* Runs for a single cycle when entering the unholding state. *)
METHOD M420_Unholding_Entry : BOOL
VAR_INPUT
END_VAR
END_METHOD

(* Runs for a single cycle when exiting the unholding state. *)
METHOD M422_Unholding_Exit : BOOL
VAR_INPUT
END_VAR
END_METHOD

(* Runs for a single cycle when entering the suspending state. *)
METHOD M500_Suspending_Entry : BOOL
VAR_INPUT
END_VAR
END_METHOD

(* Runs for a single cycle when exiting the suspending state. *)
METHOD M502_Suspending_Exit : BOOL
VAR_INPUT
END_VAR
END_METHOD

(* Runs for a single cycle when entering the unsuspending state. *)
METHOD M520_Unsuspending_Entry : BOOL
VAR_INPUT
END_VAR
END_METHOD

(* Runs for a single cycle when exiting the unsuspending state. *)
METHOD M522_Unsuspending_Exit : BOOL
VAR_INPUT
END_VAR
END_METHOD

END_INTERFACE

// Abstract/FB_StateMachine
(*
===============================================================================
State Machine
===============================================================================
:Contact: Kevin Sanita <ksanita@sensata.com>
:Last Edited: December 2021

:Description: Abstract class containing the framework for a PackML state machine

:Notes:
* Function blocks that extend this should implement the ``I_Stateful`` interface and call ``A_StateMachine``

:Change Log:
- **December 2021** Initial version
- **July 2022** Added ability to disable state methods
*)
FUNCTION_BLOCK ABSTRACT FB_StateMachine EXTENDS FB_Module IMPLEMENTS I_Stateful, I_StateControl
VAR_INPUT
	(* If this is set to true, no I_Stateful methods will be ran and all
	transition states will immediately continue to the next waiting state. *)
	in_bDisableStateMethods: BOOL := FALSE;
END_VAR
VAR_OUTPUT
END_VAR
VAR
	sm_enumState : E_PackMLState; // Current machine state	

	// Transition Variables
	sm_bAbort : BOOL; // Go directly to the aborting state from anywhere in the power on group
	sm_bStop : BOOL; // Go directly to the stopping state from anywhere in the run group
	
	sm_bAborted : BOOL; // Done aborting
	sm_bClear : BOOL; // Clear the abort state
	sm_bCleared : BOOL; // Done clearing
	sm_bStopped : BOOL; // Done stopping
	sm_bReset : BOOL; // Go to the resetting state
	
	sm_bIdle : BOOL; // Done resetting
	sm_bStart : BOOL; // Start the execution
	sm_bStarted : BOOL; // Execution started
	sm_bFinished : BOOL; // Execution finished
	sm_bCompleted : BOOL; // Done completing
	sm_bReturn : BOOL; // Return to resetting state
	
	sm_bHold : BOOL; // Hold the machine
	sm_bHeld : BOOL; // Machine is held
	sm_bUnhold : BOOL; // Unhold the machine
	sm_bUnheld : BOOL; // Machine is unheld
	
	sm_bSuspend : BOOL; // Suspend the machine
	sm_bSuspended : BOOL; // Machine is suspended
	sm_bUnsuspend : BOOL; // Unsuspend the machine
	sm_bUnsuspended : BOOL; // Machine is unsuspended
	
	// Commands to control state variables from methods
	{attribute: 'hide'}
	sm_bAbortCmd: BOOL;			// bAbort from method
	{attribute: 'hide'}
	sm_bAbortedCmd: BOOL;		// bAborted from method 
	{attribute: 'hide'}
	sm_bClearCmd: BOOL;			// bClear from method 
	{attribute: 'hide'}
	sm_bClearedCmd: BOOL;		// bCleared from method 
	{attribute: 'hide'}
	sm_bStopCmd: BOOL;			// bStop from method
	{attribute: 'hide'}
	sm_bStoppedCmd: BOOL;		// bStopped from method 
	{attribute: 'hide'}
	sm_bResetCmd: BOOL;			// bReset from method 
	{attribute: 'hide'}
	sm_bIdleCmd: BOOL;			// bIdle from method 
	{attribute: 'hide'}
	sm_bStartCmd: BOOL;			// bStart from method 
	{attribute: 'hide'}
	sm_bStartedCmd: BOOL;		// bStarted from method 
	{attribute: 'hide'}
	sm_bFinishedCmd: BOOL;		// bFinished from method 
	{attribute: 'hide'}
	sm_bHoldCmd: BOOL;			// bHold from method 
	{attribute: 'hide'}
	sm_bSuspendCmd: BOOL;		// bSuspend from method
	{attribute: 'hide'}
	sm_bCompletedCmd: BOOL;		// bCompleted from method
	{attribute: 'hide'}
	sm_bReturnCmd: BOOL;		// bReturn from method 
	{attribute: 'hide'}
	sm_bHeldCmd: BOOL;			// bHeld from method 
	{attribute: 'hide'}
	sm_bUnholdCmd: BOOL;		// bUnhold from method 
	{attribute: 'hide'}
	sm_bUnheldCmd: BOOL;		// bUnheld from method 
	{attribute: 'hide'}	
	sm_bSuspendedCmd: BOOL;		// bSuspended from method 
	{attribute: 'hide'}
	sm_bUnsuspendCmd: BOOL;		// bUnsuspend from method 
	{attribute: 'hide'}
	sm_bUnsuspendedCmd: BOOL;	// bUnsuspended from method 
END_VAR

A_StateMachine();

(* TRUE if the state machine is able to be aborted. *)
PROPERTY P_bAbortable : BOOL
GET
P_bAbortable := sm_enumState <> E_PackMLState.Aborting AND sm_enumState <> E_PackMLState.Aborted;
END_GET
END_PROPERTY

(* TRUE if the state machine is able to be stopped. *)
PROPERTY P_bStoppable : BOOL
GET
P_bStoppable := P_bAbortable
	AND sm_enumState <> E_PackMLState.Clearing
	AND sm_enumState <> E_PackMLState.Stopping
	AND sm_enumState <> E_PackMLState.Stopped;
END_GET
END_PROPERTY

(* The current E_PackMLState state of the state machine. *)
PROPERTY P_enumState : E_PackMLState
GET
P_enumState := sm_enumState;
END_GET
END_PROPERTY

(* Go directly to the abort state while in the stoppable or abortable group. *)
METHOD M_Abort : BOOL
IF THIS^.P_bAbortable THEN
	sm_bAbort := TRUE;
END_IF

IF sm_enumState = E_PackMLState.Aborted THEN
	M_Abort := TRUE;
	sm_bAbort := FALSE;
ELSE
	M_Abort := FALSE;
END_IF
END_METHOD

(* Go to the stopped state from the aborted state. *)
METHOD M_Clear : BOOL
IF sm_enumState = E_PackMLState.Aborted THEN
	sm_bClear := TRUE;
END_IF	

IF sm_enumState = E_PackMLState.Stopped THEN
	M_Clear := TRUE;
	sm_bClear := FALSE;
ELSE
	M_Clear := FALSE;
END_IF
END_METHOD

(* Go to the completing state from the execute state. *)
METHOD M_Complete : BOOL
IF sm_enumState = E_PackMLState.Execute THEN
	sm_bFinished := TRUE;
END_IF

IF sm_enumState = E_PackMLState.Complete THEN
	M_Complete := TRUE;
	sm_bFinished := FALSE;
ELSE
	M_Complete := FALSE;
END_IF
END_METHOD

(* Go to the held state from the execute state. *)
METHOD M_Hold : BOOL
IF sm_enumState = E_PackMLState.Execute THEN
	sm_bHold := TRUE;
END_IF

IF sm_enumState = E_PackMLState.Held THEN
	M_Hold := TRUE;
	sm_bHold := FALSE;
ELSE
	M_Hold := FALSE;
END_IF
END_METHOD

(* Go to the idle state from the complete or stopped state. *)
METHOD M_Reset : BOOL
IF sm_enumState = E_PackMLState.Stopped THEN
	sm_bReset := TRUE;
ELSIF sm_enumState = E_PackMLState.Complete THEN
	sm_bReturn := TRUE;
END_IF

IF sm_enumState = E_PackMLState.Idle THEN
	M_Reset := TRUE;
	sm_bReset := FALSE;
	sm_bReturn := FALSE;
ELSE
	M_Reset := FALSE;
END_IF
END_METHOD

(* Go to the execute state from the idle states. *)
METHOD M_Start : BOOL
IF sm_enumState = E_PackMLState.Idle THEN
	sm_bStart := TRUE;
END_IF

IF sm_enumState = E_PackMLState.Execute THEN
	M_Start := TRUE;
	sm_bStart := FALSE;
ELSE
	M_Start := FALSE;
END_IF
END_METHOD

(* Go to the stopped state while in the stoppable group. *)
METHOD M_Stop : BOOL
IF THIS^.P_bStoppable THEN
	sm_bStop := TRUE;
END_IF

IF sm_enumState = E_PackMLState.Stopped THEN
	M_Stop := TRUE;
	sm_bStop := FALSE;
ELSE
	M_Stop := FALSE;
END_IF
END_METHOD

(* Go to the suspended state from the execute state. *)
METHOD M_Suspend : BOOL
IF sm_enumState = E_PackMLState.Execute THEN
	sm_bSuspend := TRUE;
END_IF

IF sm_enumState = E_PackMLState.Suspended THEN
	M_Suspend := TRUE;
	sm_bSuspend := FALSE;
ELSE
	M_Suspend := FALSE;
END_IF
END_METHOD

(* Go to the execute state from the held state. *)
METHOD M_Unhold : BOOL
IF sm_enumState = E_PackMLState.Held THEN
	sm_bUnhold := TRUE;
END_IF

IF sm_enumState = E_PackMLState.Execute THEN
	M_Unhold := TRUE;
	sm_bUnhold := FALSE;
ELSE
	M_Unhold := FALSE;
END_IF
END_METHOD

(* Go to the execute state from the suspended state. *)
METHOD M_Unsuspend : BOOL
IF sm_enumState = E_PackMLState.Suspended THEN
	sm_bUnsuspend := TRUE;
END_IF

IF sm_enumState = E_PackMLState.Execute THEN
	M_Unsuspend := TRUE;
	sm_bUnsuspend := FALSE;
ELSE
	M_Unsuspend := FALSE;
END_IF
END_METHOD

ACTION A000_Aborting_Entry:
{attribute 'hide'}
sm_enumState := E_PackMLState.Aborting;
sm_bAborted := FALSE;

(* If state methods are not disabled, run the aborting entry method. *)
IF NOT in_bDisableStateMethods THEN
	THIS^.M_LogMessage('Entered $'Aborting$' state.');
	THIS^.M000_Aborting_Entry();
ELSE
	THIS^.M_LogWarning('State methods disabled! Entered $'Aborting$' state. Skipping to $'Aborted$' state...');
	sm_bAborted := TRUE;
END_IF
END_ACTION

ACTION A001_Aborting:
{attribute 'hide'}
(* If state methods are not disabled, run the aborting method. *)
IF NOT in_bDisableStateMethods THEN
	THIS^.M001_Aborting(bAborted => sm_bAbortedCmd);
	IF sm_bAbortedCmd THEN
		sm_bAborted := TRUE;
	END_IF
END_IF
END_ACTION

ACTION A002_Aborting_Exit:
{attribute 'hide'}
(* If state methods are not disabled, run the aborting exit method. *)
IF NOT in_bDisableStateMethods THEN
	THIS^.M002_Aborting_Exit();
END_IF
END_ACTION

{attribute 'hide'}
METHOD M000_Aborting_Entry : BOOL
END_METHOD

{attribute 'hide'}
METHOD M001_Aborting : BOOL
VAR_OUTPUT
	(* Move to the Aborted state*)
	bAborted	: BOOL	:= FALSE;
END_VAR
// Skip to aborted state by default
bAborted := TRUE;
END_METHOD

{attribute 'hide'}
METHOD M002_Aborting_Exit : BOOL
END_METHOD

ACTION A010_Aborted_Entry:
{attribute 'hide'}
sm_enumState := E_PackMLState.Aborted;
sm_bClear := FALSE;

(* If state methods are not disabled, run the aborted entry method. *)
IF NOT in_bDisableStateMethods THEN
	THIS^.M_LogMessage('Entered $'Aborted$' state.');
	THIS^.M010_Aborted_Entry();
ELSE
	THIS^.M_LogWarning('State methods disabled! Entered $'Aborted$' state. Waiting for transition...');
END_IF
END_ACTION

ACTION A011_Aborted:
{attribute 'hide'}
(* If state methods are enabled, run the aborted method. *)
IF NOT in_bDisableStateMethods THEN
	THIS^.M011_Aborted(bClear => sm_bClearCmd);
	IF sm_bClearCmd THEN
		sm_bClear := TRUE;
	END_IF
END_IF
END_ACTION

ACTION A012_Aborted_Exit:
{attribute 'hide'}
(* If state methods are not disabled, run the aborted exit method. *)
IF NOT in_bDisableStateMethods THEN
	THIS^.M012_Aborted_Exit();
END_IF
END_ACTION

{attribute 'hide'}
METHOD M010_Aborted_Entry : BOOL
END_METHOD

{attribute 'hide'}
METHOD M011_Aborted : BOOL
VAR_OUTPUT
	(* Move to the Clearing state*)
	bClear	: BOOL	:= FALSE;
END_VAR
END_METHOD

{attribute 'hide'}
METHOD M012_Aborted_Exit : BOOL
END_METHOD

ACTION A020_Clearing_Entry:
{attribute 'hide'}
sm_enumState := E_PackMLState.Clearing;
sm_bCleared := FALSE;
sm_bAbort := FALSE;

IF NOT in_bDisableStateMethods THEN
	THIS^.M_LogMessage('Entered $'Clearing$' state.');
	THIS^.M020_Clearing_Entry();
ELSE
	THIS^.M_LogWarning('State methods disabled! Entered $'Clearing$' state. Skipping to $'Stopped$' state...');
	sm_bCleared := TRUE;
END_IF
END_ACTION

ACTION A021_Clearing:
{attribute 'hide'}
(* If state methods are not disabled, run the clearing method. *)
IF NOT in_bDisableStateMethods THEN
	THIS^.M021_Clearing(bCleared => sm_bClearedCmd, bAbort => sm_bAbortCmd);
	IF sm_bAbortCmd THEN
		sm_bAbort := TRUE;
	ELSIF sm_bClearedCmd THEN
		sm_bCleared := TRUE;
	END_IF
END_IF
END_ACTION

ACTION A022_Clearing_Exit:
{attribute 'hide'}
IF NOT in_bDisableStateMethods THEN
	THIS^.M022_Clearing_Exit();
END_IF
END_ACTION

{attribute 'hide'}
METHOD M020_Clearing_Entry : BOOL
END_METHOD

{attribute 'hide'}
METHOD M021_Clearing : BOOL
VAR_OUTPUT
	(* Move to the Stopped state*)
	bCleared	: BOOL	:= FALSE;
	(* Move to the Aborting state*)
	bAbort		: BOOL	:= FALSE;
END_VAR
// Skip to stopped state by default
bCleared := TRUE;
END_METHOD

{attribute 'hide'}
METHOD M022_Clearing_Exit : BOOL
END_METHOD

ACTION A100_Stopping_Entry:
{attribute 'hide'}
sm_enumState := E_PackMLState.Stopping;
sm_bStopped := FALSE;

(* If state methods are not disabled, run the stopping entry method. *)
IF NOT in_bDisableStateMethods THEN
	THIS^.M_LogMessage('Entered $'Stopping$' state.');
	THIS^.M100_Stopping_Entry();
ELSE
	THIS^.M_LogWarning('State methods disabled! Entered $'Stopping$' state. Skipping to $'Stopped$' state...');
	sm_bStopped := TRUE;
END_IF
END_ACTION

ACTION A101_Stopping:
{attribute 'hide'}
(* If state methods are not disabled, run the stopping method. *)
IF NOT in_bDisableStateMethods THEN
	THIS^.M101_Stopping(bStopped => sm_bStoppedCmd, bAbort => sm_bAbortCmd);
	IF sm_bAbortCmd THEN
		sm_bAbort := TRUE;
	ELSIF sm_bStoppedCmd THEN
		sm_bStopped := TRUE;
	END_IF
END_IF
END_ACTION

ACTION A102_Stopping_Exit:
{attribute 'hide'}
(* If state methods are not disabled, run the stopping exit method. *)
IF NOT in_bDisableStateMethods THEN
	THIS^.M102_Stopping_Exit();
END_IF
END_ACTION

{attribute 'hide'}
METHOD M100_Stopping_Entry : BOOL
END_METHOD

{attribute 'hide'}
METHOD M101_Stopping : BOOL
VAR_OUTPUT
	(* Move to the Stopped state*)
	bStopped	: BOOL	:= FALSE;
	(* Move to the Aborting state*)
	bAbort		: BOOL	:= FALSE;
END_VAR
// Move to stopped state by default
bStopped := TRUE;
END_METHOD

{attribute 'hide'}
METHOD M102_Stopping_Exit : BOOL
END_METHOD

ACTION A110_Stopped_Entry:
{attribute 'hide'}
sm_enumState := E_PackMLState.Stopped;
sm_bReset := FALSE;

